C03647=1205.474,-109.246,-38.036,179.217,5.484,149.197
C03648=1205.479,-109.496,-38.027,179.214,5.484,149.197
C03649=1205.485,-109.746,-38.017,179.213,5.484,149.198
C03650=1205.489,-109.996,-38.007,179.210,5.483,149.198
C03651=1205.495,-110.246,-37.997,179.208,5.484,149.199
C03652=1205.501,-110.495,-37.987,179.205,5.483,149.200
C03653=1205.506,-110.745,-37.978,179.203,5.483,149.200
C03654=1205.512,-110.995,-37.968,179.201,5.483,149.201
C03655=1205.516,-111.244,-37.959,179.199,5.483,149.202
C03656=1205.522,-111.495,-37.949,179.196,5.482,149.202
C03657=1205.527,-111.744,-37.939,179.194,5.483,149.203
C03658=1205.532,-111.994,-37.929,179.192,5.482,149.204
C03659=1205.537,-112.244,-37.920,179.190,5.482,149.204
C03660=1205.543,-112.493,-37.910,179.187,5.482,149.205
C03661=1205.549,-112.743,-37.900,179.185,5.482,149.206
C03662=1205.553,-112.993,-37.890,179.183,5.483,149.206
C03663=1205.559,-113.243,-37.880,179.181,5.482,149.207
C03664=1205.564,-113.493,-37.871,179.179,5.482,149.208
C03665=1205.569,-113.742,-37.861,179.176,5.482,149.208
C03666=1205.575,-113.992,-37.852,179.175,5.482,149.209
C03667=1205.580,-114.242,-37.842,179.172,5.482,149.209
C03668=1205.585,-114.491,-37.833,179.170,5.482,149.210
C03669=1205.590,-114.742,-37.822,179.168,5.481,149.211
C03670=1205.596,-114.992,-37.813,179.166,5.482,149.211
C03671=1205.601,-115.241,-37.803,179.163,5.481,149.212
C03672=1205.606,-115.490,-37.794,179.161,5.482,149.213
C03673=1205.611,-115.740,-37.785,179.159,5.481,149.213
C03674=1205.617,-115.990,-37.775,179.157,5.481,149.214
C03675=1205.622,-116.240,-37.766,179.154,5.481,149.215
C03676=1205.628,-116.489,-37.755,179.152,5.481,149.215
C03677=1205.633,-116.739,-37.747,179.150,5.480,149.216
C03678=1205.639,-116.989,-37.737,179.148,5.481,149.217
C03679=1205.643,-117.239,-37.727,179.145,5.480,149.217
C03680=1205.649,-117.489,-37.718,179.143,5.480,149.218
C03681=1205.654,-117.738,-37.708,179.141,5.480,149.219
C03682=1205.659,-117.988,-37.699,179.139,5.480,149.219
C03683=1205.664,-118.238,-37.689,179.136,5.480,149.220
C03684=1205.670,-118.488,-37.680,179.134,5.480,149.220
C03685=1205.675,-118.737,-37.670,179.132,5.479,149.221
C03686=1205.680,-118.987,-37.661,179.130,5.480,149.222
C03687=1205.685,-119.237,-37.652,179.128,5.480,149.222
C03688=1205.691,-119.486,-37.642,179.126,5.479,149.223
C03689=1205.696,-119.736,-37.633,179.124,5.480,149.224
C03690=1205.702,-119.986,-37.623,179.121,5.479,149.224
C03691=1205.706,-120.236,-37.613,179.119,5.479,149.225
C03692=1205.712,-120.486,-37.604,179.117,5.479,149.226
C03693=1205.717,-120.736,-37.594,179.115,5.479,149.226
C03694=1205.722,-120.986,-37.585,179.112,5.478,149.227
C03695=1205.727,-121.235,-37.576,179.110,5.479,149.227
C03696=1205.733,-121.485,-37.566,179.108,5.478,149.228
C03697=1205.738,-121.735,-37.557,179.106,5.478,149.229
C03698=1205.743,-121.984,-37.548,179.103,5.478,149.229
C03699=1205.749,-122.234,-37.538,179.101,5.478,149.230
C03700=1205.754,-122.484,-37.529,179.099,5.478,149.231
C03701=1205.759,-122.733,-37.520,179.097,5.478,149.231
C03702=1205.765,-122.984,-37.510,179.095,5.478,149.232
C03703=1205.770,-123.233,-37.501,179.093,5.478,149.232
C03704=1205.775,-123.483,-37.492,179.091,5.478,149.233
C03705=1205.781,-123.733,-37.482,179.088,5.478,149.234
C03706=1205.786,-123.983,-37.473,179.086,5.478,149.234
C03707=1205.791,-124.232,-37.464,179.084,5.477,149.235
C03708=1205.797,-124.482,-37.454,179.082,5.478,149.236
C03709=1205.802,-124.732,-37.445,179.079,5.477,149.236
C03710=1205.807,-124.982,-37.436,179.077,5.477,149.237
C03711=1205.812,-125.231,-37.427,179.075,5.477,149.238
C03712=1205.818,-125.481,-37.417,179.073,5.477,149.238
C03713=1205.823,-125.731,-37.408,179.070,5.476,149.239
C03714=1205.828,-125.981,-37.400,179.068,5.477,149.240
C03715=1205.834,-126.230,-37.389,179.067,5.477,149.240
C03716=1205.839,-126.480,-37.380,179.064,5.476,149.241
C03717=1205.844,-126.730,-37.372,179.062,5.476,149.241
C03718=1205.423,-126.740,-37.410,179.058,5.480,149.243
C03719=1205.417,-126.491,-37.418,179.060,5.480,149.243
C03720=1205.413,-126.241,-37.428,179.063,5.480,149.242
C03721=1205.407,-125.991,-37.437,179.064,5.480,149.242
C03722=1205.402,-125.741,-37.446,179.066,5.480,149.241
C03723=1205.396,-125.491,-37.455,179.069,5.480,149.240
C03724=1205.391,-125.242,-37.465,179.071,5.480,149.240
C03725=1205.386,-124.992,-37.474,179.073,5.480,149.239
C03726=1205.380,-124.742,-37.483,179.075,5.480,149.238
C03727=1205.375,-124.492,-37.492,179.078,5.481,149.238
C03728=1205.370,-124.243,-37.502,179.080,5.480,149.237
C03729=1205.364,-123.993,-37.511,179.082,5.481,149.236
C03730=1205.359,-123.743,-37.520,179.084,5.481,149.236
C03731=1205.354,-123.494,-37.530,179.087,5.481,149.235
C03732=1205.349,-123.244,-37.539,179.088,5.481,149.235
C03733=1205.343,-122.994,-37.548,179.091,5.482,149.234
C03734=1205.338,-122.744,-37.557,179.093,5.481,149.233
C03735=1205.333,-122.495,-37.567,179.095,5.481,149.233
C03736=1205.327,-122.245,-37.576,179.097,5.482,149.232
C03737=1205.322,-121.995,-37.585,179.099,5.481,149.231
C03738=1205.317,-121.746,-37.595,179.102,5.482,149.231
C03739=1205.312,-121.495,-37.604,179.104,5.482,149.230
C03740=1205.307,-121.246,-37.614,179.106,5.482,149.229
C03741=1205.301,-120.996,-37.623,179.108,5.482,149.229
C03742=1205.296,-120.746,-37.632,179.111,5.482,149.228
C03743=1205.291,-120.497,-37.642,179.112,5.482,149.228
C03744=1205.285,-120.247,-37.651,179.115,5.483,149.227
C03745=1205.280,-119.997,-37.660,179.117,5.482,149.226
C03746=1205.275,-119.748,-37.670,179.119,5.483,149.226
C03747=1205.269,-119.498,-37.679,179.121,5.483,149.225
C03748=1205.264,-119.248,-37.689,179.124,5.483,149.224
C03749=1205.258,-118.998,-37.699,179.126,5.483,149.224
C03750=1205.253,-118.748,-37.707,179.128,5.483,149.223
C03751=1205.249,-118.498,-37.717,179.130,5.483,149.222
C03752=1205.243,-118.248,-37.727,179.132,5.483,149.222
C03753=1205.238,-117.999,-37.736,179.135,5.483,149.221
C03754=1205.232,-117.749,-37.746,179.137,5.483,149.220
C03755=1205.227,-117.500,-37.756,179.139,5.483,149.220
C03756=1205.222,-117.250,-37.765,179.141,5.484,149.219
C03757=1205.216,-117.000,-37.775,179.144,5.484,149.218
C03758=1205.211,-116.750,-37.784,179.146,5.484,149.218
C03759=1205.205,-116.500,-37.793,179.148,5.484,149.217
C03760=1205.200,-116.251,-37.803,179.150,5.484,149.217
C03761=1205.195,-116.001,-37.812,179.153,5.484,149.216
C03762=1205.190,-115.751,-37.822,179.154,5.484,149.215
C03763=1205.185,-115.501,-37.831,179.157,5.485,149.215
C03764=1205.180,-115.251,-37.841,179.159,5.484,149.214
C03765=1205.174,-115.002,-37.850,179.161,5.485,149.213
C03766=1205.169,-114.752,-37.860,179.163,5.485,149.213
C03767=1205.164,-114.503,-37.870,179.166,5.485,149.212
C03768=1205.158,-114.253,-37.880,179.168,5.485,149.212
C03769=1205.153,-114.003,-37.889,179.170,5.486,149.211
C03770=1205.148,-113.753,-37.899,179.172,5.485,149.210
C03771=1205.143,-113.503,-37.909,179.175,5.486,149.209
C03772=1205.137,-113.253,-37.918,179.177,5.486,149.209
C03773=1205.132,-113.004,-37.928,179.179,5.486,149.208
C03774=1205.126,-112.754,-37.937,179.181,5.486,149.207
C03775=1205.121,-112.505,-37.947,179.184,5.486,149.207
C03776=1205.116,-112.255,-37.957,179.186,5.486,149.206
C03777=1205.111,-112.004,-37.966,179.188,5.486,149.206
C03778=1205.106,-111.755,-37.976,179.190,5.486,149.205
C03779=1205.100,-111.505,-37.986,179.193,5.487,149.204
C03780=1205.095,-111.255,-37.996,179.195,5.486,149.204
C03781=1205.089,-111.006,-38.006,179.197,5.486,149.203
C03782=1205.084,-110.756,-38.015,179.199,5.487,149.202
C03783=1205.079,-110.506,-38.025,179.201,5.486,149.202
C03784=1205.074,-110.257,-38.035,179.204,5.487,149.201
C03785=1205.068,-110.006,-38.044,179.205,5.487,149.201
C03786=1205.064,-109.757,-38.054,179.208,5.487,149.200
C03787=1205.058,-109.508,-38.064,179.210,5.487,149.199
C03788=1205.052,-109.258,-38.074,179.212,5.488,149.199
C03789=1205.048,-109.008,-38.084,179.214,5.487,149.198
C03790=1205.042,-108.758,-38.094,179.217,5.488,149.197
C03791=1205.037,-108.508,-38.103,179.219,5.487,149.196
C03792=1205.031,-108.259,-38.113,179.221,5.488,149.196
C03793=1205.026,-108.009,-38.123,179.223,5.488,149.195
C03794=1205.021,-107.759,-38.132,179.226,5.488,149.195
C03795=1205.016,-107.509,-38.143,179.228,5.488,149.194
C03796=1205.011,-107.260,-38.152,179.230,5.488,149.193
C03797=1205.005,-107.010,-38.162,179.233,5.488,149.193
C03798=1205.000,-106.759,-38.172,179.235,5.488,149.192
C03799=1204.995,-106.510,-38.182,179.237,5.488,149.191
C03800=1204.989,-106.261,-38.192,179.239,5.489,149.191
C03801=1204.984,-106.010,-38.202,179.242,5.489,149.190
C03802=1204.979,-105.760,-38.212,179.244,5.489,149.190
C03803=1204.974,-105.511,-38.222,179.246,5.489,149.189
C03804=1204.968,-105.261,-38.232,179.249,5.489,149.188
C03805=1204.963,-105.012,-38.242,179.251,5.489,149.187
C03806=1204.957,-104.762,-38.251,179.253,5.490,149.187
C03807=1204.953,-104.512,-38.261,179.255,5.489,149.186
C03808=1204.947,-104.263,-38.271,179.258,5.490,149.185
C03809=1204.942,-104.013,-38.282,179.260,5.489,149.185
C03810=1204.937,-103.763,-38.292,179.262,5.490,149.184
C03811=1204.932,-103.513,-38.301,179.264,5.490,149.184
C03812=1204.926,-103.263,-38.311,179.267,5.490,149.183
C03813=1204.920,-103.014,-38.321,179.269,5.490,149.182
C03814=1204.916,-102.764,-38.331,179.271,5.491,149.182
C03815=1204.911,-102.514,-38.342,179.273,5.490,149.181
C03816=1204.905,-102.265,-38.352,179.276,5.491,149.180
C03817=1204.901,-102.015,-38.362,179.278,5.491,149.180
C03818=1204.895,-101.765,-38.371,179.280,5.491,149.179
C03819=1204.889,-101.493,-38.383,179.283,5.491,149.178
C03820=1204.883,-101.222,-38.393,179.285,5.491,149.178
C03821=1204.878,-100.951,-38.404,179.287,5.492,149.177
C03822=1204.872,-100.680,-38.416,179.290,5.492,149.176
C03823=1204.867,-100.430,-38.426,179.292,5.492,149.175
C03824=1204.861,-100.180,-38.435,179.295,5.492,149.175
C03825=1204.856,-99.930,-38.446,179.296,5.492,149.174
C03826=1204.851,-99.680,-38.456,179.299,5.492,149.174
C03827=1204.846,-99.431,-38.465,179.301,5.492,149.173
C03828=1204.841,-99.181,-38.476,179.304,5.492,149.172
C03829=1204.835,-98.931,-38.486,179.305,5.492,149.172
C03830=1204.830,-98.682,-38.496,179.308,5.493,149.171
C03831=1204.825,-98.432,-38.507,179.310,5.492,149.170
C03832=1204.820,-98.182,-38.517,179.313,5.493,149.170
C03833=1204.814,-97.933,-38.527,179.314,5.493,149.169
C03834=1204.809,-97.683,-38.537,179.317,5.493,149.168
C03835=1204.804,-97.433,-38.548,179.319,5.493,149.168
C03836=1204.798,-97.183,-38.558,179.322,5.493,149.167
C03837=1204.794,-96.934,-38.568,179.324,5.493,149.166
C03838=1204.788,-96.684,-38.578,179.326,5.494,149.166
C03839=1204.783,-96.434,-38.588,179.328,5.493,149.165
C03840=1204.778,-96.184,-38.599,179.331,5.494,149.164
C03841=1204.772,-95.935,-38.609,179.333,5.494,149.164
C03842=1204.766,-95.685,-38.619,179.335,5.494,149.163
C03843=1204.761,-95.435,-38.630,179.338,5.495,149.162
C03844=1204.756,-95.186,-38.639,179.340,5.494,149.162
C03845=1204.751,-94.935,-38.650,179.342,5.495,149.161
C03846=1204.746,-94.686,-38.660,179.344,5.495,149.160
C03847=1204.740,-94.436,-38.670,179.347,5.495,149.160
C03848=1204.735,-94.186,-38.681,179.349,5.495,149.159
C03849=1204.730,-93.937,-38.691,179.351,5.496,149.159
C03850=1204.725,-93.687,-38.702,179.353,5.495,149.158
C03851=1204.720,-93.438,-38.712,179.356,5.496,149.157
C03852=1204.715,-93.188,-38.722,179.358,5.495,149.156
C03853=1204.710,-92.938,-38.733,179.360,5.496,149.156
C03854=1204.704,-92.688,-38.743,179.362,5.496,149.155
C03855=1204.699,-92.438,-38.754,179.365,5.496,149.155
C03856=1204.693,-92.189,-38.764,179.367,5.496,149.154
C03857=1204.688,-91.939,-38.774,179.370,5.496,149.153
C03858=1204.683,-91.689,-38.785,179.372,5.497,149.153
C03859=1204.677,-91.440,-38.796,179.374,5.496,149.152
C03860=1204.672,-91.190,-38.806,179.377,5.497,149.151
C03861=1204.667,-90.940,-38.816,179.379,5.497,149.150
C03862=1204.662,-90.690,-38.827,179.381,5.497,149.150
C03863=1204.656,-90.440,-38.837,179.383,5.497,149.149
C03864=1204.651,-90.191,-38.847,179.386,5.497,149.149
C03865=1204.647,-89.941,-38.858,179.388,5.497,149.148
C03866=1204.641,-89.692,-38.868,179.390,5.498,149.147
C03867=1204.636,-89.442,-38.879,179.392,5.497,149.147
C03868=1204.631,-89.192,-38.889,179.395,5.498,149.146
C03869=1204.626,-88.942,-38.900,179.397,5.497,149.145
C03870=1204.620,-88.693,-38.910,179.400,5.498,149.145
C03871=1204.615,-88.443,-38.921,179.402,5.499,149.144
C03872=1204.610,-88.193,-38.931,179.404,5.498,149.143
C03873=1204.605,-87.943,-38.942,179.406,5.499,149.143
C03874=1204.599,-87.694,-38.953,179.409,5.498,149.142
C03875=1204.594,-87.444,-38.963,179.411,5.499,149.141
C03876=1204.589,-87.194,-38.974,179.413,5.499,149.141
C03877=1204.584,-86.945,-38.985,179.416,5.499,149.140
C03878=1204.578,-86.695,-38.995,179.418,5.499,149.139
C03879=1204.573,-86.445,-39.006,179.420,5.499,149.139
C03880=1204.568,-86.195,-39.016,179.422,5.499,149.138
C03881=1204.563,-85.946,-39.027,179.425,5.500,149.137
C03882=1204.558,-85.696,-39.037,179.427,5.500,149.137
C03883=1204.553,-85.446,-39.048,179.429,5.500,149.136
C03884=1204.547,-85.197,-39.059,179.432,5.500,149.135
C03885=1204.542,-84.947,-39.069,179.434,5.500,149.135
C03886=1204.536,-84.697,-39.080,179.436,5.501,149.134
C03887=1204.531,-84.447,-39.092,179.438,5.500,149.133
C03888=1204.526,-84.198,-39.102,179.441,5.501,149.133
C03889=1204.521,-83.947,-39.112,179.443,5.500,149.132
C03890=1204.515,-83.698,-39.123,179.445,5.501,149.131
C03891=1204.510,-83.448,-39.134,179.448,5.502,149.131
C03892=1204.505,-83.199,-39.144,179.450,5.501,149.130
C03893=1204.500,-82.949,-39.155,179.453,5.502,149.129
C03894=1204.494,-82.699,-39.166,179.454,5.502,149.129
C03895=1204.490,-82.450,-39.177,179.457,5.502,149.128
C03896=1204.484,-82.200,-39.187,179.459,5.502,149.127
C03897=1204.479,-81.950,-39.198,179.462,5.502,149.127
C03898=1204.474,-81.700,-39.209,179.464,5.503,149.126
C03899=1204.468,-81.451,-39.220,179.466,5.503,149.126
C03900=1204.463,-81.201,-39.231,179.469,5.503,149.125
C03901=1204.458,-80.951,-39.241,179.471,5.503,149.124
C03902=1204.453,-80.702,-39.252,179.473,5.503,149.123
C03903=1204.448,-80.452,-39.263,179.476,5.503,149.123
C03904=1204.443,-80.203,-39.274,179.478,5.504,149.122
C03905=1204.437,-79.952,-39.285,179.480,5.503,149.122
C03906=1204.432,-79.703,-39.295,179.482,5.504,149.121
C03907=1204.427,-79.453,-39.307,179.485,5.504,149.120
C03908=1204.421,-79.203,-39.317,179.487,5.504,149.119
C03909=1204.417,-78.954,-39.328,179.489,5.504,149.119
C03910=1204.412,-78.703,-39.339,179.491,5.504,149.118
C03911=1204.406,-78.454,-39.350,179.494,5.504,149.118
C03912=1204.401,-78.204,-39.361,179.496,5.504,149.117
C03913=1204.395,-77.955,-39.372,179.499,5.505,149.116
C03914=1204.390,-77.705,-39.382,179.501,5.505,149.116
C03915=1204.386,-77.455,-39.394,179.503,5.505,149.115
C03916=1204.380,-77.206,-39.405,179.506,5.505,149.114
C03917=1204.375,-76.956,-39.416,179.508,5.505,149.113
C03918=1204.369,-76.707,-39.427,179.511,5.506,149.113
C03919=1204.364,-76.457,-39.437,179.513,5.506,149.112
C03920=1204.359,-76.207,-39.449,179.515,5.506,149.112
C03921=1204.353,-75.957,-39.459,179.518,5.506,149.111
C03922=1204.349,-75.707,-39.471,179.520,5.506,149.110
C03923=1204.343,-75.436,-39.483,179.522,5.506,149.109
C03924=1204.337,-75.166,-39.495,179.525,5.507,149.109
C03925=1204.332,-74.896,-39.506,179.527,5.507,149.108
C03926=1204.326,-74.625,-39.518,179.530,5.507,149.107
C03927=1204.321,-74.375,-39.529,179.532,5.507,149.107
C03928=1204.315,-74.125,-39.541,179.534,5.507,149.106
C03929=1204.310,-73.876,-39.552,179.537,5.507,149.105
C03930=1204.305,-73.626,-39.562,179.539,5.507,149.105
C03931=1204.300,-73.376,-39.573,179.541,5.508,149.104
C03932=1204.294,-73.127,-39.585,179.544,5.508,149.103
C03933=1204.289,-72.877,-39.596,179.546,5.508,149.103
C03934=1204.284,-72.627,-39.607,179.549,5.508,149.102
C03935=1204.278,-72.378,-39.618,179.550,5.508,149.101
C03936=1204.273,-72.128,-39.629,179.553,5.509,149.101
C03937=1204.269,-71.878,-39.640,179.556,5.509,149.100
C03938=1204.263,-71.629,-39.652,179.558,5.509,149.099
C03939=1204.258,-71.379,-39.662,179.561,5.509,149.099
C03940=1204.253,-71.129,-39.674,179.563,5.509,149.098
C03941=1204.248,-70.879,-39.686,179.565,5.510,149.097
C03942=1204.242,-70.630,-39.696,179.567,5.510,149.097
C03943=1204.237,-70.380,-39.707,179.570,5.510,149.096
C03944=1204.232,-70.130,-39.719,179.572,5.510,149.095
C03945=1204.227,-69.881,-39.730,179.574,5.510,149.095
C03946=1204.222,-69.631,-39.741,179.577,5.510,149.094
C03947=1204.216,-69.381,-39.752,179.579,5.511,149.093
C03948=1204.211,-69.131,-39.764,179.581,5.511,149.093
C03949=1204.205,-68.882,-39.775,179.584,5.511,149.092
C03950=1204.201,-68.632,-39.786,179.586,5.511,149.091
C03951=1204.196,-68.382,-39.797,179.589,5.511,149.091
C03952=1204.190,-68.133,-39.808,179.591,5.512,149.090
C03953=1204.185,-67.883,-39.820,179.593,5.512,149.089
C03954=1204.180,-67.633,-39.832,179.596,5.512,149.089
C03955=1204.175,-67.384,-39.843,179.598,5.512,149.088
C03956=1204.169,-67.134,-39.853,179.600,5.512,149.087
C03957=1204.164,-66.884,-39.865,179.603,5.513,149.087
C03958=1204.159,-66.635,-39.876,179.605,5.513,149.086
C03959=1204.154,-66.385,-39.888,179.607,5.513,149.085
C03960=1204.149,-66.135,-39.900,179.609,5.513,149.085
C03961=1204.143,-65.886,-39.911,179.612,5.513,149.084
C03962=1204.138,-65.636,-39.922,179.615,5.514,149.083
C03963=1204.133,-65.386,-39.933,179.617,5.513,149.083
C03964=1204.128,-65.136,-39.945,179.619,5.514,149.082
C03965=1204.123,-64.887,-39.956,179.621,5.514,149.081
C03966=1204.117,-64.637,-39.968,179.624,5.514,149.081
C03967=1204.113,-64.387,-39.979,179.626,5.515,149.080
C03968=1204.107,-64.138,-39.991,179.628,5.514,149.079
C03969=1204.102,-63.888,-40.002,179.631,5.515,149.079
C03970=1204.096,-63.639,-40.014,179.633,5.516,149.078
C03971=1204.092,-63.389,-40.025,179.635,5.515,149.077
C03972=1204.086,-63.139,-40.037,179.638,5.516,149.077
C03973=1204.082,-62.889,-40.048,179.640,5.515,149.076
C03974=1204.076,-62.640,-40.060,179.643,5.516,149.075
C03975=1204.071,-62.391,-40.071,179.646,5.516,149.075
C03976=1204.065,-62.141,-40.083,179.647,5.516,149.074
C03977=1204.061,-61.891,-40.094,179.650,5.517,149.073
C03978=1204.055,-61.640,-40.105,179.652,5.517,149.073
C03979=1204.050,-61.391,-40.116,179.655,5.517,149.072
C03980=1204.045,-61.141,-40.128,179.657,5.517,149.071
C03981=1204.040,-60.892,-40.139,179.659,5.517,149.071
C03982=1204.034,-60.643,-40.152,179.661,5.518,149.070
C03983=1204.030,-60.393,-40.163,179.664,5.518,149.069
C03984=1204.024,-60.143,-40.175,179.666,5.518,149.069
C03985=1204.019,-59.893,-40.187,179.669,5.518,149.068
C03986=1204.014,-59.644,-40.198,179.672,5.519,149.067
C03987=1204.009,-59.394,-40.210,179.674,5.518,149.067
C03988=1204.003,-59.145,-40.221,179.676,5.519,149.066
C03989=1203.998,-58.895,-40.233,179.678,5.519,149.065
C03990=1203.993,-58.645,-40.244,179.681,5.519,149.065
C03991=1203.988,-58.395,-40.256,179.683,5.520,149.064
C03992=1203.982,-58.145,-40.268,179.685,5.519,149.063
C03993=1203.978,-57.896,-40.279,179.688,5.520,149.063
C03994=1203.972,-57.646,-40.291,179.691,5.520,149.062
C03995=1203.968,-57.396,-40.302,179.692,5.520,149.061
C03996=1203.962,-57.146,-40.314,179.695,5.521,149.061
C03997=1203.957,-56.898,-40.327,179.698,5.521,149.060
C03998=1203.952,-56.648,-40.338,179.700,5.521,149.059
C03999=1203.946,-56.398,-40.350,179.702,5.521,149.059
C04000=1203.942,-56.148,-40.361,179.704,5.521,149.058
C04001=1203.936,-55.898,-40.373,179.707,5.522,149.057
C04002=1203.931,-55.648,-40.385,179.709,5.522,149.057
C04003=1203.926,-55.399,-40.396,179.711,5.522,149.056
C04004=1203.921,-55.150,-40.409,179.714,5.522,149.055
C04005=1203.916,-54.900,-40.421,179.717,5.523,149.055
C04006=1203.911,-54.650,-40.432,179.719,5.522,149.054
C04007=1203.905,-54.400,-40.444,179.721,5.523,149.053
C04008=1203.900,-54.150,-40.456,179.724,5.524,149.053
C04009=1203.896,-53.901,-40.468,179.726,5.523,149.052
C04010=1203.890,-53.651,-40.480,179.728,5.524,149.051
C04011=1203.884,-53.402,-40.491,179.731,5.524,149.051
C04012=1203.880,-53.152,-40.502,179.733,5.524,149.050
C04013=1203.874,-52.903,-40.515,179.736,5.524,149.049
C04014=1203.869,-52.653,-40.527,179.738,5.525,149.049
C04015=1203.864,-52.403,-40.539,179.740,5.525,149.048
C04016=1203.859,-52.153,-40.550,179.743,5.525,149.047
C04017=1203.854,-51.904,-40.563,179.745,5.526,149.047
C04018=1203.848,-51.654,-40.574,179.747,5.525,149.046
C04019=1203.844,-51.405,-40.586,179.750,5.526,149.045
C04020=1203.838,-51.155,-40.598,179.753,5.526,149.044
C04021=1203.833,-50.905,-40.610,179.754,5.526,149.044
C04022=1203.828,-50.655,-40.622,179.757,5.527,149.043
C04023=1203.822,-50.405,-40.634,179.759,5.526,149.043
C04024=1203.818,-50.156,-40.646,179.762,5.527,149.042
C04025=1203.812,-49.907,-40.658,179.764,5.527,149.041
C04026=1203.807,-49.657,-40.670,179.767,5.527,149.040
C04027=1203.802,-49.386,-40.683,179.769,5.527,149.040
C04028=1203.796,-49.117,-40.696,179.772,5.528,149.039
C04029=1203.791,-48.847,-40.709,179.775,5.528,149.038
C04030=1203.785,-48.576,-40.722,179.777,5.529,149.038
C04031=1203.780,-48.327,-40.734,179.779,5.528,149.037
C04032=1203.775,-48.077,-40.747,179.782,5.529,149.036
C04033=1203.769,-47.827,-40.758,179.785,5.529,149.036
C04034=1203.764,-47.577,-40.770,179.786,5.529,149.035
C04035=1203.760,-47.328,-40.782,179.789,5.530,149.034
C04036=1203.754,-47.078,-40.794,179.792,5.530,149.034
C04037=1203.749,-46.829,-40.807,179.794,5.530,149.033
C04038=1203.744,-46.579,-40.819,179.796,5.530,149.032
C04039=1203.738,-46.329,-40.831,179.799,5.531,149.032
C04040=1203.733,-46.080,-40.843,179.801,5.531,149.031
C04041=1203.728,-45.830,-40.854,179.803,5.531,149.030
C04042=1203.723,-45.581,-40.867,179.806,5.532,149.030
C04043=1203.718,-45.331,-40.879,179.808,5.531,149.029
C04044=1203.713,-45.082,-40.892,179.811,5.532,149.028
C04045=1203.707,-44.832,-40.903,179.813,5.532,149.028
C04046=1203.702,-44.582,-40.916,179.816,5.533,149.027
C04047=1203.697,-44.333,-40.928,179.818,5.533,149.026
C04048=1203.692,-44.083,-40.940,179.820,5.533,149.026
C04049=1203.686,-43.833,-40.952,179.823,5.534,149.025
C04050=1203.682,-43.584,-40.965,179.825,5.533,149.024
C04051=1203.677,-43.334,-40.977,179.828,5.534,149.024
C04052=1203.672,-43.084,-40.989,179.830,5.534,149.023
C04053=1203.666,-42.834,-41.001,179.832,5.534,149.022
C04054=1203.661,-42.585,-41.014,179.835,5.534,149.021
C04055=1203.656,-42.335,-41.026,179.837,5.535,149.021
C04056=1203.651,-42.086,-41.038,179.839,5.535,149.020
C04057=1203.645,-41.836,-41.050,179.842,5.535,149.020
C04058=1203.640,-41.587,-41.063,179.845,5.536,149.019
C04059=1203.635,-41.337,-41.075,179.847,5.536,149.018
C04060=1203.630,-41.087,-41.088,179.849,5.536,149.017
C04061=1203.625,-40.837,-41.100,179.852,5.536,149.017
C04062=1203.620,-40.587,-41.112,179.854,5.537,149.016
C04063=1203.615,-40.338,-41.125,179.856,5.537,149.016
C04064=1203.609,-40.089,-41.137,179.859,5.537,149.015
C04065=1203.604,-39.839,-41.149,179.862,5.538,149.014
C04066=1203.599,-39.589,-41.162,179.864,5.538,149.014
C04067=1203.593,-39.340,-41.174,179.866,5.538,149.013
C04068=1203.589,-39.089,-41.187,179.869,5.538,149.012
C04069=1203.584,-38.840,-41.199,179.871,5.539,149.012
C04070=1203.578,-38.590,-41.211,179.873,5.539,149.011
C04071=1203.573,-38.341,-41.224,179.876,5.539,149.010
C04072=1203.568,-38.092,-41.236,179.879,5.540,149.010
C04073=1203.563,-37.842,-41.248,179.881,5.540,149.009
C04074=1203.558,-37.592,-41.261,179.883,5.540,149.008
C04075=1203.553,-37.342,-41.274,179.886,5.541,149.007
C04076=1203.548,-37.092,-41.286,179.888,5.541,149.007
C04077=1203.542,-36.843,-41.298,179.890,5.541,149.006
C04078=1203.537,-36.594,-41.311,179.893,5.541,149.006
C04079=1203.532,-36.344,-41.323,179.896,5.542,149.005
C04080=1203.527,-36.094,-41.336,179.898,5.542,149.004
C04081=1203.522,-35.844,-41.348,179.900,5.542,149.003
C04082=1203.517,-35.595,-41.361,179.903,5.543,149.003
C04083=1203.512,-35.346,-41.373,179.905,5.543,149.002
C04084=1203.507,-35.096,-41.385,179.907,5.543,149.002
C04085=1203.502,-34.846,-41.398,179.910,5.544,149.001
C04086=1203.496,-34.596,-41.412,179.913,5.544,149.000
C04087=1203.491,-34.347,-41.424,179.915,5.544,149.000
C04088=1203.486,-34.097,-41.436,179.917,5.544,148.999
C04089=1203.481,-33.848,-41.449,179.920,5.545,148.998
C04090=1203.476,-33.598,-41.462,179.922,5.545,148.998
C04091=1203.471,-33.348,-41.474,179.924,5.545,148.997
C04092=1203.466,-33.099,-41.487,179.927,5.546,148.996
C04093=1203.461,-32.850,-41.499,179.930,5.546,148.996
C04094=1203.455,-32.599,-41.512,179.932,5.546,148.995
C04095=1203.450,-32.349,-41.525,179.934,5.546,148.994
C04096=1203.445,-32.100,-41.537,179.937,5.547,148.993
C04097=1203.440,-31.851,-41.550,179.939,5.547,148.993
C04098=1203.435,-31.601,-41.563,179.941,5.547,148.992
C04099=1203.430,-31.351,-41.576,179.944,5.548,148.992
C04100=1203.425,-31.102,-41.588,179.947,5.548,148.991
C04101=1203.419,-30.852,-41.601,179.949,5.548,148.990
C04102=1203.414,-30.602,-41.614,179.951,5.548,148.989
C04103=1203.409,-30.353,-41.626,179.954,5.549,148.989
C04104=1203.404,-30.103,-41.639,179.957,5.549,148.988
C04105=1203.399,-29.854,-41.651,179.958,5.549,148.988
C04106=1203.394,-29.604,-41.665,179.961,5.550,148.987
C04107=1203.388,-29.354,-41.678,179.963,5.550,148.986
C04108=1203.383,-29.105,-41.690,179.966,5.551,148.986
C04109=1203.379,-28.855,-41.703,179.968,5.550,148.985
C04110=1203.374,-28.606,-41.716,179.971,5.551,148.984
C04111=1203.368,-28.356,-41.729,179.974,5.551,148.983
C04112=1203.363,-28.107,-41.742,179.976,5.552,148.983
C04113=1203.358,-27.857,-41.755,179.978,5.552,148.982
C04114=1203.353,-27.607,-41.767,179.980,5.552,148.982
C04115=1203.347,-27.358,-41.780,179.983,5.553,148.981
C04116=1203.343,-27.108,-41.793,179.986,5.553,148.980
C04117=1203.338,-26.858,-41.806,179.988,5.553,148.979
C04118=1203.332,-26.609,-41.818,179.991,5.553,148.979
C04119=1203.327,-26.359,-41.832,179.993,5.554,148.978
C04120=1203.322,-26.109,-41.845,179.995,5.555,148.978
C04121=1203.317,-25.860,-41.857,179.997,5.554,148.977
C04122=1203.312,-25.610,-41.871,-180.000,5.555,148.976
C04123=1203.307,-25.360,-41.883,-179.997,5.555,148.976
C04124=1203.301,-25.111,-41.896,-179.995,5.556,148.975
C04125=1203.297,-24.861,-41.909,-179.993,5.555,148.974
C04126=1203.291,-24.612,-41.922,-179.990,5.556,148.974
C04127=1203.286,-24.362,-41.935,-179.988,5.557,148.973
C04128=1203.281,-24.112,-41.948,-179.985,5.557,148.972
C04129=1203.276,-23.863,-41.962,-179.983,5.557,148.972
C04130=1203.271,-23.613,-41.975,-179.980,5.557,148.971
C04131=1203.265,-23.344,-41.989,-179.978,5.558,148.970
C04132=1203.260,-23.074,-42.002,-179.975,5.558,148.970
C04133=1203.254,-22.804,-42.016,-179.972,5.559,148.969
C04134=1203.249,-22.536,-42.031,-179.970,5.559,148.968
C04135=1203.244,-22.285,-42.044,-179.967,5.560,148.967
C04136=1203.239,-22.036,-42.057,-179.965,5.559,148.967
C04137=1203.234,-21.786,-42.070,-179.962,5.560,148.966
C04138=1203.228,-21.536,-42.083,-179.960,5.560,148.965
C04139=1203.223,-21.288,-42.096,-179.957,5.561,148.965
C04140=1203.218,-21.037,-42.110,-179.955,5.561,148.964
C04141=1203.213,-20.788,-42.122,-179.953,5.561,148.963
C04142=1203.208,-20.538,-42.135,-179.950,5.562,148.963
C04143=1203.203,-20.288,-42.148,-179.947,5.562,148.962
C04144=1203.198,-20.040,-42.162,-179.945,5.562,148.961
C04145=1203.193,-19.789,-42.175,-179.943,5.562,148.961
C04146=1203.187,-19.540,-42.188,-179.940,5.563,148.960
C04147=1203.183,-19.290,-42.201,-179.938,5.564,148.960
C04148=1203.177,-19.041,-42.215,-179.935,5.564,148.959
C04149=1203.172,-18.792,-42.227,-179.933,5.564,148.958
C04150=1203.167,-18.541,-42.241,-179.930,5.564,148.957
C04151=1203.162,-18.292,-42.254,-179.928,5.565,148.957
C04152=1203.157,-18.042,-42.268,-179.925,5.565,148.956
C04153=1203.152,-17.793,-42.280,-179.923,5.565,148.955
C04154=1203.146,-17.543,-42.294,-179.921,5.566,148.955
C04155=1203.142,-17.294,-42.307,-179.918,5.566,148.954
C04156=1203.136,-17.044,-42.321,-179.916,5.567,148.954
C04157=1203.131,-16.794,-42.334,-179.913,5.567,148.953
C04158=1203.126,-16.545,-42.348,-179.911,5.567,148.952
C04159=1203.121,-16.295,-42.360,-179.908,5.567,148.951
C04160=1203.116,-16.045,-42.374,-179.905,5.568,148.951
C04161=1203.111,-15.796,-42.387,-179.903,5.569,148.950
C04162=1203.105,-15.547,-42.400,-179.901,5.569,148.950
C04163=1203.101,-15.297,-42.413,-179.899,5.569,148.949
C04164=1203.095,-15.048,-42.427,-179.896,5.569,148.948
C04165=1203.091,-14.798,-42.440,-179.893,5.570,148.947
C04166=1203.085,-14.548,-42.454,-179.891,5.570,148.947
C04167=1203.081,-14.299,-42.467,-179.888,5.571,148.946
C04168=1203.075,-14.049,-42.480,-179.886,5.571,148.946
C04169=1203.070,-13.800,-42.494,-179.884,5.571,148.945
C04170=1203.065,-13.550,-42.507,-179.881,5.572,148.944
C04171=1203.060,-13.300,-42.521,-179.878,5.572,148.944
C04172=1203.055,-13.050,-42.535,-179.876,5.573,148.943
C04173=1203.050,-12.801,-42.547,-179.874,5.573,148.942
C04174=1203.045,-12.551,-42.561,-179.871,5.573,148.941
C04175=1203.039,-12.302,-42.575,-179.869,5.574,148.941
C04176=1203.035,-12.052,-42.588,-179.866,5.574,148.940
C04177=1203.029,-11.802,-42.601,-179.863,5.575,148.940
C04178=1203.025,-11.553,-42.615,-179.861,5.575,148.939
C04179=1203.019,-11.303,-42.628,-179.859,5.575,148.938
C04180=1203.014,-11.054,-42.643,-179.856,5.575,148.938
C04181=1203.009,-10.804,-42.655,-179.853,5.576,148.937
C04182=1203.004,-10.555,-42.669,-179.851,5.577,148.936
C04183=1202.999,-10.305,-42.682,-179.849,5.577,148.936
C04184=1202.994,-10.056,-42.696,-179.847,5.577,148.935
C04185=1202.989,-9.805,-42.710,-179.844,5.577,148.934
C04186=1202.984,-9.557,-42.723,-179.841,5.578,148.934
C04187=1202.979,-9.307,-42.738,-179.839,5.578,148.933
C04188=1202.973,-9.057,-42.751,-179.836,5.579,148.932
C04189=1202.969,-8.808,-42.764,-179.834,5.579,148.932
C04190=1202.964,-8.558,-42.778,-179.832,5.579,148.931
C04191=1202.958,-8.309,-42.792,-179.829,5.580,148.930
C04192=1202.953,-8.059,-42.805,-179.826,5.580,148.930
C04193=1202.948,-7.810,-42.819,-179.824,5.581,148.929
C04194=1202.943,-7.560,-42.833,-179.821,5.581,148.928
C04195=1202.938,-7.310,-42.846,-179.819,5.581,148.928
C04196=1202.933,-7.061,-42.860,-179.817,5.582,148.927
C04197=1202.928,-6.811,-42.874,-179.814,5.582,148.926
C04198=1202.923,-6.562,-42.887,-179.812,5.583,148.926
C04199=1202.918,-6.312,-42.901,-179.809,5.583,148.925
C04200=1202.913,-6.062,-42.915,-179.806,5.584,148.924
C04201=1202.907,-5.813,-42.929,-179.804,5.584,148.924
C04202=1202.903,-5.563,-42.942,-179.802,5.584,148.923
C04203=1202.898,-5.314,-42.956,-179.799,5.585,148.923
C04204=1202.892,-5.064,-42.970,-179.797,5.585,148.922
C04205=1202.887,-4.814,-42.984,-179.794,5.586,148.921
C04206=1202.883,-4.565,-42.998,-179.791,5.586,148.921
C04207=1202.877,-4.315,-43.011,-179.789,5.586,148.920
C04208=1202.872,-4.066,-43.025,-179.787,5.587,148.919
C04209=1202.866,-3.817,-43.039,-179.784,5.587,148.919
C04210=1202.862,-3.567,-43.053,-179.782,5.588,148.918
C04211=1202.857,-3.317,-43.066,-179.779,5.588,148.917
C04212=1202.851,-3.068,-43.080,-179.776,5.589,148.917
C04213=1202.846,-2.818,-43.094,-179.774,5.589,148.916
C04214=1202.842,-2.568,-43.109,-179.772,5.589,148.915
C04215=1202.836,-2.319,-43.121,-179.769,5.590,148.915
C04216=1202.831,-2.069,-43.136,-179.767,5.590,148.914
C04217=1202.826,-1.820,-43.150,-179.764,5.591,148.913
C04218=1202.822,-1.570,-43.164,-179.762,5.591,148.913
C04219=1202.816,-1.321,-43.178,-179.759,5.592,148.912
C04220=1202.811,-1.071,-43.191,-179.757,5.592,148.911
C04221=1202.807,-0.821,-43.205,-179.754,5.592,148.911
C04222=1202.801,-0.572,-43.219,-179.752,5.593,148.910
C04223=1202.796,-0.322,-43.234,-179.749,5.594,148.909
C04224=1202.791,-0.073,-43.248,-179.747,5.594,148.909
C04225=1202.785,0.176,-43.262,-179.744,5.595,148.908
C04226=1202.780,0.427,-43.275,-179.741,5.595,148.907
C04227=1202.776,0.676,-43.289,-179.739,5.595,148.907
C04228=1202.771,0.926,-43.303,-179.737,5.596,148.906
C04229=1202.765,1.175,-43.317,-179.735,5.596,148.906
C04230=1202.761,1.424,-43.331,-179.732,5.597,148.905
C04231=1202.756,1.674,-43.346,-179.729,5.597,148.904
C04232=1202.751,1.924,-43.360,-179.727,5.598,148.904
C04233=1202.745,2.173,-43.374,-179.724,5.598,148.903
C04234=1202.740,2.423,-43.388,-179.721,5.599,148.902
C04235=1202.735,2.692,-43.403,-179.719,5.599,148.901
C04236=1202.729,2.961,-43.418,-179.716,5.600,148.901
C04237=1202.724,3.230,-43.434,-179.713,5.600,148.900
C04238=1202.718,3.499,-43.448,-179.711,5.601,148.899
C04239=1202.713,3.749,-43.463,-179.708,5.601,148.899
C04240=1202.708,3.998,-43.477,-179.706,5.601,148.898
C04241=1202.703,4.248,-43.491,-179.704,5.602,148.898
C04242=1202.698,4.498,-43.506,-179.701,5.602,148.897
C04243=1202.693,4.747,-43.520,-179.699,5.603,148.896
C04244=1202.688,4.996,-43.534,-179.696,5.603,148.895
C04245=1202.683,5.246,-43.548,-179.693,5.604,148.895
C04246=1202.678,5.496,-43.562,-179.691,5.604,148.894
C04247=1202.672,5.745,-43.576,-179.688,5.605,148.894
C04248=1202.667,5.995,-43.591,-179.686,5.605,148.893
C04249=1202.662,6.244,-43.605,-179.684,5.605,148.892
C04250=1202.657,6.494,-43.619,-179.681,5.606,148.892
C04251=1202.652,6.744,-43.633,-179.678,5.606,148.891
C04252=1202.648,6.993,-43.648,-179.676,5.607,148.890
C04253=1202.642,7.242,-43.662,-179.674,5.608,148.890
C04254=1202.637,7.492,-43.677,-179.671,5.608,148.889
C04255=1202.632,7.741,-43.691,-179.668,5.609,148.888
C04256=1202.627,7.991,-43.705,-179.666,5.609,148.888
C04257=1202.622,8.241,-43.719,-179.663,5.610,148.887
C04258=1202.618,8.490,-43.734,-179.661,5.610,148.887
C04259=1202.612,8.739,-43.748,-179.659,5.610,148.886
C04260=1202.607,8.989,-43.762,-179.656,5.611,148.885
C04261=1202.602,9.238,-43.777,-179.653,5.611,148.885
C04262=1202.597,9.488,-43.791,-179.651,5.612,148.884
C04263=1202.592,9.738,-43.805,-179.648,5.612,148.883
C04264=1202.587,9.987,-43.820,-179.646,5.613,148.883
C04265=1202.583,10.237,-43.834,-179.643,5.613,148.882
C04266=1202.577,10.486,-43.848,-179.641,5.614,148.881
C04267=1202.572,10.735,-43.863,-179.638,5.614,148.881
C04268=1202.567,10.985,-43.878,-179.635,5.615,148.880
C04269=1202.562,11.235,-43.892,-179.633,5.615,148.879
C04270=1202.557,11.485,-43.906,-179.631,5.616,148.879
C04271=1202.552,11.734,-43.921,-179.628,5.616,148.878
C04272=1202.547,11.983,-43.936,-179.626,5.617,148.877
C04273=1202.542,12.233,-43.950,-179.623,5.617,148.877
C04274=1202.537,12.483,-43.964,-179.621,5.618,148.876
C04275=1202.531,12.732,-43.979,-179.618,5.618,148.876
C04276=1202.526,12.981,-43.994,-179.616,5.619,148.875
C04277=1202.521,13.231,-44.008,-179.613,5.619,148.874
C04278=1202.516,13.481,-44.022,-179.610,5.620,148.874
C04279=1202.512,13.730,-44.037,-179.608,5.620,148.873
C04280=1202.507,13.979,-44.051,-179.605,5.621,148.872
C04281=1202.501,14.229,-44.066,-179.604,5.621,148.872
C04282=1202.496,14.479,-44.081,-179.601,5.622,148.871
C04283=1202.491,14.728,-44.096,-179.598,5.622,148.870
C04284=1202.486,14.978,-44.110,-179.596,5.623,148.870
C04285=1202.482,15.227,-44.125,-179.593,5.623,148.869
C04286=1202.476,15.477,-44.140,-179.590,5.624,148.868
C04287=1202.471,15.727,-44.154,-179.588,5.624,148.868
C04288=1202.467,15.976,-44.169,-179.585,5.625,148.867
C04289=1202.462,16.226,-44.183,-179.583,5.625,148.866
C04290=1202.456,16.475,-44.197,-179.580,5.626,148.866
C04291=1202.451,16.724,-44.213,-179.578,5.626,148.865
C04292=1202.446,16.974,-44.227,-179.575,5.627,148.865
C04293=1202.441,17.223,-44.242,-179.573,5.628,148.864
C04294=1202.436,17.473,-44.256,-179.570,5.628,148.863
C04295=1202.430,17.723,-44.271,-179.567,5.629,148.863
C04296=1202.426,17.972,-44.286,-179.565,5.629,148.862
C04297=1202.421,18.221,-44.300,-179.563,5.629,148.861
C04298=1202.415,18.471,-44.316,-179.561,5.630,148.861
C04299=1202.410,18.720,-44.330,-179.558,5.630,148.860
C04300=1202.406,18.970,-44.345,-179.555,5.631,148.859
C04301=1202.401,19.219,-44.360,-179.553,5.632,148.859
C04302=1202.395,19.469,-44.375,-179.550,5.632,148.858
C04303=1202.391,19.718,-44.389,-179.548,5.633,148.858
C04304=1202.386,19.967,-44.404,-179.545,5.633,148.857
C04305=1202.380,20.217,-44.419,-179.542,5.634,148.856
C04306=1202.376,20.467,-44.434,-179.540,5.634,148.856
C04307=1202.371,20.716,-44.449,-179.537,5.635,148.855
C04308=1202.365,20.966,-44.464,-179.535,5.636,148.854
C04309=1202.361,21.216,-44.479,-179.532,5.636,148.854
C04310=1202.356,21.465,-44.494,-179.530,5.637,148.853
C04311=1202.350,21.715,-44.509,-179.527,5.637,148.852
C04312=1202.346,21.964,-44.524,-179.524,5.638,148.852
C04313=1202.341,22.213,-44.539,-179.522,5.639,148.851
C04314=1202.335,22.463,-44.554,-179.520,5.639,148.851
C04315=1202.331,22.712,-44.569,-179.517,5.640,148.850
C04316=1202.325,22.963,-44.583,-179.514,5.640,148.849
C04317=1202.321,23.212,-44.598,-179.512,5.641,148.849
C04318=1202.316,23.461,-44.613,-179.510,5.642,148.848
C04319=1202.310,23.711,-44.628,-179.507,5.642,148.847
C04320=1202.306,23.960,-44.643,-179.505,5.642,148.847
C04321=1202.300,24.209,-44.659,-179.502,5.642,148.846
C04322=1202.295,24.459,-44.673,-179.500,5.643,148.845
C04323=1202.291,24.708,-44.688,-179.497,5.644,148.845
C04324=1202.286,24.958,-44.704,-179.495,5.644,148.844
C04325=1202.281,25.208,-44.718,-179.492,5.645,148.844
C04326=1202.275,25.457,-44.734,-179.489,5.645,148.843
C04327=1202.271,25.706,-44.749,-179.487,5.646,148.842
C04328=1202.265,25.956,-44.764,-179.485,5.647,148.842
C04329=1202.260,26.205,-44.779,-179.482,5.647,148.841
C04330=1202.255,26.455,-44.794,-179.479,5.648,148.840
C04331=1202.250,26.705,-44.809,-179.477,5.648,148.840
C04332=1202.245,26.954,-44.824,-179.474,5.649,148.839
C04333=1202.241,27.204,-44.840,-179.472,5.650,148.839
C04334=1202.235,27.453,-44.855,-179.469,5.650,148.838
C04335=1202.230,27.703,-44.869,-179.467,5.651,148.837
C04336=1202.225,27.952,-44.885,-179.464,5.651,148.837
C04337=1202.220,28.201,-44.900,-179.461,5.652,148.836
C04338=1202.215,28.451,-44.916,-179.459,5.653,148.835
C04339=1202.210,28.720,-44.931,-179.457,5.653,148.835
C04340=1202.204,28.988,-44.948,-179.453,5.655,148.834
C04341=1202.199,29.257,-44.964,-179.451,5.655,148.833
C04342=1202.193,29.525,-44.981,-179.448,5.656,148.833
C04343=1202.189,29.776,-44.996,-179.445,5.656,148.832
C04344=1202.184,30.025,-45.011,-179.443,5.657,148.831
C04345=1202.178,30.275,-45.027,-179.440,5.657,148.831
C04346=1202.174,30.524,-45.042,-179.438,5.658,148.830
C04347=1202.168,30.773,-45.057,-179.435,5.659,148.830
C04348=1202.164,31.022,-45.072,-179.433,5.659,148.829
C04349=1202.159,31.272,-45.088,-179.430,5.660,148.828
C04350=1202.154,31.522,-45.103,-179.427,5.660,148.828
C04351=1202.149,31.771,-45.118,-179.425,5.661,148.827
C04352=1202.143,32.021,-45.134,-179.423,5.662,148.826
C04353=1202.139,32.270,-45.149,-179.420,5.662,148.826
C04354=1202.134,32.520,-45.165,-179.417,5.663,148.825
C04355=1202.129,32.769,-45.180,-179.415,5.663,148.825
C04356=1202.124,33.018,-45.195,-179.412,5.664,148.824
C04357=1202.118,33.268,-45.211,-179.410,5.664,148.823
C04358=1202.114,33.518,-45.226,-179.407,5.665,148.823
C04359=1202.109,33.767,-45.242,-179.405,5.666,148.822
C04360=1202.103,34.016,-45.258,-179.402,5.666,148.821
C04361=1202.099,34.265,-45.273,-179.400,5.667,148.821
C04362=1202.094,34.516,-45.288,-179.397,5.667,148.820
C04363=1202.089,34.765,-45.304,-179.394,5.668,148.819
C04364=1202.084,35.014,-45.319,-179.392,5.669,148.819
C04365=1202.079,35.263,-45.335,-179.390,5.669,148.818
C04366=1202.074,35.514,-45.351,-179.387,5.670,148.818
C04367=1202.069,35.763,-45.366,-179.384,5.670,148.817
C04368=1202.064,36.012,-45.381,-179.382,5.671,148.816
C04369=1202.058,36.261,-45.397,-179.380,5.672,148.816
C04370=1202.054,36.511,-45.412,-179.377,5.672,148.815
C04371=1202.049,36.761,-45.428,-179.374,5.673,148.814
C04372=1202.044,37.010,-45.443,-179.372,5.673,148.814
C04373=1202.038,37.259,-45.459,-179.370,5.674,148.813
C04374=1202.034,37.509,-45.474,-179.367,5.675,148.813
C04375=1202.029,37.759,-45.490,-179.364,5.676,148.812
C04376=1202.024,38.007,-45.506,-179.361,5.677,148.811
C04377=1202.019,38.258,-45.522,-179.359,5.678,148.811
C04378=1202.014,38.507,-45.537,-179.356,5.678,148.810
C04379=1202.009,38.756,-45.553,-179.354,5.679,148.810
C04380=1202.003,39.005,-45.568,-179.351,5.679,148.809
C04381=1201.999,39.256,-45.584,-179.349,5.680,148.808
C04382=1201.994,39.505,-45.599,-179.346,5.681,148.808
C04383=1201.989,39.753,-45.615,-179.343,5.681,148.807
C04384=1201.984,40.004,-45.631,-179.341,5.682,148.806
C04385=1201.979,40.253,-45.647,-179.339,5.683,148.806
C04386=1201.973,40.502,-45.663,-179.336,5.683,148.805
C04387=1201.969,40.752,-45.678,-179.333,5.684,148.805
C04388=1201.964,41.002,-45.694,-179.331,5.684,148.804
C04389=1201.959,41.250,-45.710,-179.328,5.685,148.803
C04390=1201.954,41.500,-45.726,-179.326,5.686,148.803
C04391=1201.949,41.750,-45.741,-179.323,5.686,148.802
C04392=1201.943,41.999,-45.757,-179.321,5.687,148.801
C04393=1201.940,42.248,-45.773,-179.318,5.687,148.801
C04394=1201.934,42.498,-45.789,-179.315,5.689,148.800
C04395=1201.929,42.748,-45.805,-179.313,5.689,148.800
C04396=1201.924,42.997,-45.820,-179.310,5.690,148.799
C04397=1201.919,43.246,-45.837,-179.307,5.690,148.798
C04398=1201.914,43.496,-45.852,-179.305,5.691,148.798
C04399=1201.909,43.746,-45.868,-179.303,5.692,148.797
C04400=1201.904,43.994,-45.884,-179.300,5.692,148.797
C04401=1201.900,44.244,-45.900,-179.297,5.693,148.796
C04402=1201.894,44.494,-45.915,-179.295,5.694,148.795
C04403=1201.890,44.743,-45.932,-179.293,5.694,148.795
C04404=1201.884,44.992,-45.948,-179.290,5.695,148.794
C04405=1201.879,45.242,-45.963,-179.288,5.696,148.794
C04406=1201.875,45.491,-45.980,-179.285,5.696,148.793
C04407=1201.869,45.741,-45.995,-179.282,5.698,148.792
C04408=1201.865,45.990,-46.012,-179.279,5.698,148.792
C04409=1201.859,46.240,-46.028,-179.277,5.699,148.791
C04410=1201.854,46.490,-46.044,-179.274,5.700,148.791
C04411=1201.849,46.739,-46.060,-179.272,5.700,148.790
C04412=1201.844,46.988,-46.076,-179.269,5.701,148.789
C04413=1201.840,47.237,-46.092,-179.267,5.702,148.789
C04414=1201.834,47.487,-46.108,-179.264,5.702,148.788
C04415=1201.829,47.737,-46.124,-179.262,5.703,148.787
C04416=1201.824,47.986,-46.140,-179.259,5.703,148.787
C04417=1201.820,48.236,-46.155,-179.257,5.704,148.786
C04418=1201.815,48.484,-46.172,-179.254,5.705,148.786
C04419=1201.810,48.734,-46.188,-179.251,5.706,148.785
C04420=1201.805,48.983,-46.204,-179.248,5.707,148.784
C04421=1201.801,49.233,-46.220,-179.246,5.707,148.784
C04422=1201.795,49.482,-46.237,-179.244,5.708,148.783
C04423=1201.790,49.732,-46.253,-179.241,5.709,148.783
C04424=1201.785,49.981,-46.269,-179.239,5.709,148.782
C04425=1201.780,50.231,-46.285,-179.236,5.710,148.781
C04426=1201.775,50.480,-46.301,-179.234,5.710,148.781
C04427=1201.770,50.730,-46.317,-179.231,5.711,148.780
C04428=1201.765,50.979,-46.334,-179.228,5.713,148.780
C04429=1201.761,51.229,-46.350,-179.226,5.713,148.779
C04430=1201.755,51.478,-46.366,-179.223,5.714,148.778
C04431=1201.751,51.727,-46.382,-179.221,5.715,148.778
C04432=1201.745,51.977,-46.398,-179.218,5.715,148.777
C04433=1201.741,52.226,-46.415,-179.216,5.716,148.777
C04434=1201.736,52.475,-46.431,-179.213,5.716,148.776
C04435=1201.731,52.725,-46.447,-179.211,5.717,148.775
C04436=1201.726,52.974,-46.463,-179.208,5.718,148.775
C04437=1201.721,53.224,-46.479,-179.205,5.719,148.774
C04438=1201.715,53.473,-46.496,-179.202,5.720,148.773
C04439=1201.711,53.723,-46.513,-179.200,5.721,148.773
C04440=1201.705,53.972,-46.528,-179.198,5.721,148.772
C04441=1201.701,54.222,-46.545,-179.195,5.722,148.772
C04442=1201.696,54.470,-46.561,-179.193,5.723,148.771
C04443=1201.691,54.739,-46.579,-179.190,5.724,148.771
C04444=1201.685,55.008,-46.597,-179.187,5.724,148.770
C04445=1201.680,55.277,-46.614,-179.184,5.725,148.769
C04446=1201.675,55.545,-46.632,-179.182,5.726,148.769
C04447=1201.670,55.794,-46.649,-179.178,5.727,148.768
C04448=1201.665,56.044,-46.664,-179.176,5.728,148.767
C04449=1201.660,56.293,-46.682,-179.174,5.728,148.767
C04450=1201.655,56.542,-46.698,-179.171,5.729,148.766
C04451=1201.650,56.792,-46.715,-179.168,5.729,148.765
C04452=1201.645,57.041,-46.730,-179.166,5.730,148.765
C04453=1201.640,57.291,-46.747,-179.164,5.731,148.764
C04454=1201.635,57.540,-46.764,-179.160,5.732,148.764
C04455=1201.630,57.789,-46.781,-179.158,5.733,148.763
C04456=1201.625,58.039,-46.796,-179.156,5.734,148.763
C04457=1201.621,58.289,-46.813,-179.153,5.734,148.762
C04458=1201.616,58.537,-46.829,-179.151,5.735,148.761
C04459=1201.610,58.787,-46.847,-179.148,5.736,148.761
C04460=1201.605,59.036,-46.863,-179.146,5.736,148.760
C04461=1201.601,59.286,-46.880,-179.142,5.738,148.759
C04462=1201.595,59.536,-46.896,-179.140,5.738,148.759
C04463=1201.590,59.785,-46.913,-179.138,5.739,148.758
C04464=1201.586,60.034,-46.929,-179.135,5.740,148.758
C04465=1201.581,60.284,-46.946,-179.133,5.740,148.757
C04466=1201.575,60.533,-46.963,-179.130,5.741,148.757
C04467=1201.571,60.782,-46.979,-179.127,5.742,148.756
C04468=1201.566,61.032,-46.996,-179.125,5.743,148.756
C04469=1201.561,61.281,-47.013,-179.122,5.744,148.755
C04470=1201.556,61.530,-47.030,-179.120,5.744,148.754
C04471=1201.552,61.780,-47.046,-179.117,5.745,148.754
C04472=1201.546,62.029,-47.063,-179.115,5.746,148.753
C04473=1201.541,62.278,-47.080,-179.112,5.747,148.752
C04474=1201.537,62.529,-47.096,-179.109,5.748,148.752
C04475=1201.531,62.778,-47.113,-179.107,5.749,148.751
C04476=1201.526,63.027,-47.129,-179.104,5.749,148.751
C04477=1201.522,63.277,-47.146,-179.102,5.750,148.750
C04478=1201.516,63.526,-47.163,-179.099,5.751,148.750
C04479=1201.512,63.775,-47.180,-179.096,5.752,148.749
C04480=1201.507,64.025,-47.196,-179.094,5.753,148.748
C04481=1201.502,64.274,-47.214,-179.091,5.753,148.748
C04482=1201.497,64.523,-47.231,-179.089,5.754,148.747
C04483=1201.492,64.772,-47.248,-179.086,5.755,148.746
C04484=1201.487,65.022,-47.265,-179.083,5.756,148.746
C04485=1201.482,65.271,-47.281,-179.081,5.757,148.745
C04486=1201.477,65.520,-47.298,-179.078,5.757,148.745
C04487=1201.473,65.770,-47.315,-179.076,5.758,148.744
C04488=1201.467,66.020,-47.332,-179.073,5.759,148.744
C04489=1201.462,66.269,-47.348,-179.071,5.759,148.743
C04490=1201.458,66.518,-47.365,-179.068,5.761,148.743
C04491=1201.453,66.768,-47.382,-179.065,5.762,148.742
C04492=1201.448,67.017,-47.399,-179.063,5.762,148.741
C04493=1201.443,67.266,-47.417,-179.061,5.763,148.741
C04494=1201.438,67.515,-47.433,-179.058,5.764,148.740
C04495=1201.433,67.765,-47.451,-179.055,5.765,148.739
C04496=1201.428,68.015,-47.467,-179.053,5.766,148.739
C04497=1201.423,68.264,-47.484,-179.050,5.767,148.738
C04498=1201.418,68.513,-47.501,-179.047,5.767,148.738
C04499=1201.413,68.762,-47.519,-179.045,5.768,148.737
C04500=1201.409,69.012,-47.535,-179.042,5.769,148.737
C04501=1201.403,69.262,-47.553,-179.039,5.770,148.736
C04502=1201.399,69.511,-47.569,-179.037,5.771,148.736
C04503=1201.393,69.760,-47.586,-179.035,5.771,148.735
C04504=1201.389,70.009,-47.604,-179.032,5.773,148.734
C04505=1201.384,70.259,-47.621,-179.029,5.774,148.734
C04506=1201.379,70.508,-47.638,-179.027,5.774,148.733
C04507=1201.374,70.758,-47.655,-179.024,5.775,148.733
C04508=1201.369,71.006,-47.672,-179.022,5.776,148.732
C04509=1201.364,71.256,-47.689,-179.019,5.777,148.731
C04510=1201.360,71.506,-47.706,-179.016,5.778,148.731
C04511=1201.355,71.755,-47.724,-179.014,5.778,148.730
C04512=1201.350,72.004,-47.741,-179.011,5.779,148.730
C04513=1201.345,72.254,-47.758,-179.009,5.781,148.729
C04514=1201.339,72.503,-47.775,-179.006,5.781,148.729
C04515=1201.335,72.752,-47.792,-179.003,5.782,148.728
C04516=1201.330,73.002,-47.809,-179.001,5.783,148.727
C04517=1201.325,73.252,-47.827,-178.998,5.783,148.727
C04518=1201.320,73.500,-47.844,-178.996,5.785,148.726
C04519=1201.315,73.750,-47.861,-178.993,5.786,148.726
C04520=1201.311,73.999,-47.879,-178.991,5.786,148.725
C04521=1201.305,74.248,-47.895,-178.988,5.787,148.725
C04522=1201.300,74.498,-47.913,-178.985,5.788,148.724
C04523=1201.296,74.747,-47.930,-178.983,5.789,148.723
C04524=1201.291,74.997,-47.947,-178.980,5.790,148.723
C04525=1201.286,75.246,-47.965,-178.978,5.791,148.722
C04526=1201.281,75.495,-47.982,-178.975,5.792,148.722
C04527=1201.276,75.744,-48.000,-178.972,5.793,148.721
C04528=1201.271,75.994,-48.017,-178.970,5.793,148.720
C04529=1201.267,76.244,-48.034,-178.968,5.794,148.720
C04530=1201.262,76.493,-48.052,-178.964,5.796,148.719
C04531=1201.256,76.742,-48.069,-178.962,5.796,148.719
C04532=1201.252,76.991,-48.086,-178.960,5.797,148.718
C04533=1201.246,77.241,-48.103,-178.957,5.798,148.718
C04534=1201.242,77.490,-48.121,-178.954,5.799,148.717
C04535=1201.236,77.740,-48.139,-178.952,5.800,148.717
C04536=1201.232,77.988,-48.156,-178.949,5.801,148.716
C04537=1201.227,78.238,-48.173,-178.947,5.801,148.715
C04538=1201.222,78.487,-48.191,-178.944,5.803,148.715
C04539=1201.217,78.737,-48.209,-178.941,5.803,148.714
C04540=1201.213,78.986,-48.226,-178.939,5.804,148.714
C04541=1201.208,79.235,-48.244,-178.936,5.805,148.713
C04542=1201.203,79.485,-48.261,-178.934,5.807,148.713
C04543=1201.198,79.734,-48.279,-178.931,5.807,148.712
C04544=1201.193,79.984,-48.296,-178.928,5.808,148.711
C04545=1201.188,80.233,-48.314,-178.926,5.809,148.711
C04546=1201.183,80.482,-48.332,-178.923,5.810,148.710
C04547=1201.178,80.751,-48.351,-178.920,5.811,148.710
C04548=1201.172,81.019,-48.370,-178.917,5.812,148.709
C04549=1201.167,81.287,-48.388,-178.915,5.813,148.709
C04550=1201.162,81.556,-48.408,-178.912,5.814,148.708
C04551=1201.157,81.805,-48.424,-178.909,5.815,148.707
C04552=1201.152,82.054,-48.442,-178.907,5.816,148.707
C04553=1201.147,82.303,-48.460,-178.905,5.816,148.706
C04554=1201.142,82.553,-48.478,-178.901,5.818,148.706
C04555=1201.137,82.802,-48.496,-178.899,5.819,148.705
C04556=1201.132,83.052,-48.514,-178.897,5.819,148.704
C04557=1201.128,83.300,-48.531,-178.894,5.821,148.704
C04558=1201.123,83.550,-48.548,-178.891,5.821,148.703
C04559=1201.118,83.799,-48.566,-178.889,5.822,148.703
C04560=1201.113,84.049,-48.584,-178.886,5.823,148.702
C04561=1201.108,84.298,-48.602,-178.883,5.824,148.702
C04562=1201.103,84.548,-48.619,-178.881,5.825,148.701
C04563=1201.098,84.797,-48.637,-178.879,5.826,148.701
C04564=1201.093,85.046,-48.655,-178.876,5.828,148.700
C04565=1201.088,85.295,-48.673,-178.873,5.828,148.700
C04566=1201.083,85.544,-48.691,-178.871,5.829,148.699
C04567=1201.080,85.794,-48.708,-178.868,5.830,148.698
C04568=1201.075,86.044,-48.726,-178.865,5.831,148.698
C04569=1201.070,86.293,-48.744,-178.863,5.832,148.697
C04570=1201.065,86.542,-48.762,-178.860,5.833,148.697
C04571=1201.060,86.791,-48.780,-178.857,5.834,148.696
C04572=1201.055,87.040,-48.798,-178.855,5.835,148.696
C04573=1201.050,87.290,-48.815,-178.853,5.835,148.695
C04574=1201.045,87.539,-48.833,-178.850,5.837,148.695
C04575=1201.040,87.789,-48.851,-178.847,5.838,148.694
C04576=1201.035,88.038,-48.869,-178.845,5.839,148.693
C04577=1201.030,88.287,-48.887,-178.842,5.840,148.693
C04578=1201.026,88.537,-48.906,-178.839,5.841,148.692
C04579=1201.021,88.786,-48.924,-178.837,5.841,148.692
C04580=1201.016,89.035,-48.942,-178.834,5.843,148.691
C04581=1201.011,89.284,-48.960,-178.832,5.844,148.691
C04582=1201.006,89.533,-48.978,-178.829,5.844,148.690
C04583=1201.001,89.783,-48.996,-178.826,5.846,148.690
C04584=1200.996,90.032,-49.014,-178.824,5.847,148.689
C04585=1200.991,90.281,-49.032,-178.821,5.847,148.688
C04586=1200.987,90.531,-49.050,-178.818,5.849,148.688
C04587=1200.982,90.780,-49.068,-178.816,5.850,148.687
C04588=1200.977,91.029,-49.086,-178.814,5.850,148.687
C04589=1200.972,91.278,-49.104,-178.811,5.852,148.686
C04590=1200.967,91.528,-49.122,-178.808,5.853,148.686
C04591=1200.962,91.777,-49.140,-178.806,5.853,148.685
C04592=1200.958,92.027,-49.159,-178.803,5.855,148.685
C04593=1200.953,92.276,-49.177,-178.800,5.856,148.684
C04594=1200.948,92.525,-49.195,-178.798,5.856,148.683
C04595=1200.943,92.774,-49.213,-178.795,5.858,148.683
C04596=1200.938,93.024,-49.231,-178.792,5.859,148.682
C04597=1200.933,93.273,-49.249,-178.790,5.859,148.682
C04598=1200.929,93.523,-49.267,-178.787,5.861,148.681
C04599=1200.924,93.772,-49.285,-178.785,5.862,148.681
C04600=1200.918,94.021,-49.304,-178.782,5.862,148.680
C04601=1200.913,94.271,-49.322,-178.780,5.864,148.680
C04602=1200.909,94.520,-49.341,-178.777,5.865,148.679
C04603=1200.904,94.769,-49.359,-178.774,5.866,148.679
C04604=1200.899,95.018,-49.377,-178.772,5.867,148.678
C04605=1200.894,95.267,-49.395,-178.769,5.868,148.677
C04606=1200.889,95.517,-49.413,-178.766,5.869,148.677
C04607=1200.884,95.767,-49.431,-178.764,5.870,148.676
C04608=1200.880,96.015,-49.450,-178.762,5.871,148.676
C04609=1200.875,96.264,-49.468,-178.758,5.872,148.675
C04610=1200.870,96.514,-49.486,-178.756,5.873,148.675
C04611=1200.865,96.764,-49.505,-178.754,5.874,148.674
C04612=1200.860,97.013,-49.523,-178.751,5.875,148.674
C04613=1200.855,97.261,-49.542,-178.748,5.876,148.673
C04614=1200.851,97.511,-49.560,-178.746,5.878,148.673
C04615=1200.845,97.761,-49.579,-178.743,5.878,148.672
C04616=1200.841,98.009,-49.597,-178.741,5.879,148.672
C04617=1200.836,98.259,-49.615,-178.738,5.881,148.671
C04618=1200.831,98.508,-49.633,-178.736,5.882,148.671
C04619=1200.826,98.758,-49.652,-178.733,5.882,148.670
C04620=1200.821,99.006,-49.671,-178.730,5.884,148.669
C04621=1200.817,99.256,-49.689,-178.728,5.885,148.669
C04622=1200.812,99.506,-49.707,-178.725,5.886,148.668
C04623=1200.807,99.754,-49.727,-178.722,5.887,148.668
C04624=1200.802,100.004,-49.745,-178.720,5.887,148.667
C04625=1200.798,100.253,-49.763,-178.717,5.889,148.667
C04626=1200.792,100.502,-49.782,-178.714,5.890,148.666
C04627=1200.787,100.752,-49.800,-178.712,5.892,148.666
C04628=1200.783,101.000,-49.819,-178.709,5.892,148.665
C04629=1200.778,101.250,-49.838,-178.707,5.893,148.665
C04630=1200.773,101.499,-49.856,-178.704,5.894,148.664
C04631=1200.768,101.748,-49.874,-178.702,5.895,148.664
C04632=1200.763,101.998,-49.893,-178.698,5.897,148.663
C04633=1200.759,102.247,-49.912,-178.696,5.898,148.663
C04634=1200.754,102.497,-49.930,-178.694,5.898,148.662
C04635=1200.749,102.746,-49.949,-178.691,5.900,148.662
C04636=1200.744,102.995,-49.968,-178.688,5.901,148.661
C04637=1200.740,103.245,-49.986,-178.686,5.902,148.661
C04638=1200.734,103.493,-50.005,-178.683,5.903,148.660
C04639=1200.729,103.743,-50.023,-178.681,5.904,148.659
C04640=1200.725,103.992,-50.043,-178.678,5.905,148.659
C04641=1200.720,104.241,-50.061,-178.676,5.906,148.658
C04642=1200.715,104.490,-50.080,-178.672,5.908,148.658
C04643=1200.710,104.740,-50.099,-178.670,5.909,148.657
C04644=1200.705,104.989,-50.117,-178.668,5.909,148.657
C04645=1200.700,105.239,-50.136,-178.665,5.911,148.656
C04646=1200.696,105.487,-50.155,-178.662,5.911,148.656
C04647=1200.690,105.736,-50.174,-178.660,5.913,148.655
C04648=1200.686,105.986,-50.193,-178.657,5.914,148.655
C04649=1200.682,106.235,-50.211,-178.654,5.916,148.654
C04650=1200.677,106.485,-50.230,-178.652,5.916,148.654
C04651=1200.671,106.753,-50.251,-178.649,5.918,148.653
C04652=1200.666,107.021,-50.270,-178.646,5.918,148.653
C04653=1200.661,107.290,-50.291,-178.643,5.920,148.652
C04654=1200.655,107.558,-50.311,-178.641,5.921,148.651
C04655=1200.651,107.808,-50.331,-178.638,5.922,148.651
C04656=1200.646,108.056,-50.350,-178.636,5.923,148.650
C04657=1200.641,108.306,-50.368,-178.633,5.925,148.650
C04658=1200.636,108.555,-50.387,-178.631,5.925,148.649
C04659=1200.632,108.804,-50.406,-178.627,5.927,148.649
C04660=1200.627,109.054,-50.425,-178.625,5.928,148.648
C04661=1200.622,109.302,-50.444,-178.622,5.929,148.648
C04662=1200.617,109.552,-50.463,-178.620,5.930,148.647
C04663=1200.613,109.801,-50.482,-178.617,5.931,148.647
C04664=1200.608,110.051,-50.501,-178.615,5.933,148.646
C04665=1200.602,110.300,-50.520,-178.612,5.933,148.646
C04666=1200.598,110.549,-50.539,-178.609,5.935,148.645
C04667=1200.593,110.798,-50.559,-178.607,5.936,148.645
C04668=1200.589,111.048,-50.577,-178.604,5.937,148.644
C04669=1200.583,111.296,-50.596,-178.602,5.938,148.644
C04670=1200.579,111.546,-50.615,-178.599,5.940,148.643
C04671=1200.574,111.795,-50.635,-178.597,5.940,148.643
C04672=1200.569,112.045,-50.654,-178.593,5.942,148.642
C04673=1200.564,112.293,-50.672,-178.591,5.943,148.642
C04674=1200.559,112.543,-50.692,-178.589,5.943,148.641
C04675=1200.554,112.792,-50.711,-178.586,5.945,148.641
C04676=1200.550,113.041,-50.730,-178.584,5.946,148.640
C04677=1200.545,113.290,-50.750,-178.581,5.948,148.640
C04678=1200.540,113.539,-50.769,-178.578,5.948,148.639
C04679=1200.535,113.789,-50.787,-178.575,5.950,148.639
C04680=1200.530,114.038,-50.807,-178.573,5.951,148.638
C04681=1200.525,114.287,-50.826,-178.570,5.952,148.638
C04682=1200.521,114.536,-50.845,-178.568,5.953,148.637
C04683=1200.516,114.785,-50.865,-178.565,5.955,148.636
C04684=1200.511,115.035,-50.884,-178.563,5.956,148.636
C04685=1200.507,115.284,-50.903,-178.560,5.957,148.636
C04686=1200.502,115.533,-50.923,-178.557,5.958,148.635
C04687=1200.497,115.782,-50.942,-178.555,5.960,148.635
C04688=1200.492,116.031,-50.961,-178.552,5.960,148.634
C04689=1200.487,116.281,-50.981,-178.549,5.962,148.634
C04690=1200.482,116.529,-51.000,-178.547,5.963,148.633
C04691=1200.477,116.779,-51.020,-178.544,5.964,148.633
C04692=1200.473,117.028,-51.039,-178.542,5.965,148.632
C04693=1200.468,117.277,-51.058,-178.539,5.967,148.632
C04694=1200.463,117.527,-51.078,-178.536,5.968,148.631
C04695=1200.458,117.776,-51.097,-178.533,5.969,148.630
C04696=1200.453,118.025,-51.116,-178.531,5.970,148.630
C04697=1200.449,118.274,-51.136,-178.528,5.971,148.629
C04698=1200.444,118.523,-51.155,-178.526,5.972,148.629
C04699=1200.439,118.773,-51.174,-178.523,5.974,148.629
C04700=1200.434,119.022,-51.194,-178.521,5.975,148.628
C04701=1200.429,119.271,-51.213,-178.518,5.976,148.628
C04702=1200.425,119.521,-51.233,-178.515,5.977,148.627
C04703=1200.420,119.769,-51.252,-178.513,5.979,148.627
C04704=1200.415,120.019,-51.271,-178.510,5.980,148.626
C04705=1200.410,120.268,-51.292,-178.507,5.981,148.626
C04706=1200.405,120.517,-51.311,-178.505,5.982,148.625
C04707=1200.400,120.766,-51.331,-178.502,5.984,148.625
C04708=1200.396,121.016,-51.350,-178.500,5.984,148.624
C04709=1200.391,121.264,-51.369,-178.497,5.986,148.624
C04710=1200.386,121.514,-51.389,-178.495,5.987,148.623
C04711=1200.382,121.763,-51.409,-178.492,5.989,148.623
C04712=1200.377,122.012,-51.428,-178.489,5.989,148.622
C04713=1200.372,122.261,-51.448,-178.487,5.991,148.622
C04714=1200.367,122.511,-51.468,-178.484,5.992,148.621
C04715=1200.362,122.760,-51.487,-178.481,5.993,148.621
C04716=1200.358,123.009,-51.507,-178.479,5.994,148.620
C04717=1200.353,123.258,-51.526,-178.476,5.996,148.620
C04718=1200.349,123.508,-51.546,-178.474,5.997,148.619
C04719=1200.343,123.757,-51.565,-178.471,5.998,148.619
C04720=1200.339,124.005,-51.586,-178.468,6.000,148.618
C04721=1200.334,124.255,-51.605,-178.466,6.001,148.618
C04722=1200.329,124.504,-51.625,-178.463,6.002,148.617
C04723=1200.324,124.753,-51.645,-178.461,6.003,148.617
C04724=1200.319,125.002,-51.665,-178.458,6.005,148.616
C04725=1200.315,125.252,-51.684,-178.455,6.005,148.616
C04726=1200.310,125.500,-51.704,-178.453,6.007,148.615
C04727=1200.305,125.750,-51.724,-178.450,6.008,148.615
C04728=1200.300,125.999,-51.744,-178.447,6.010,148.614
C04729=1200.296,126.248,-51.764,-178.445,6.011,148.614
C04730=1200.290,126.497,-51.783,-178.442,6.012,148.613
C04731=1200.286,126.747,-51.803,-178.439,6.014,148.613
C04732=1200.281,126.996,-51.823,-178.437,6.015,148.612
C04733=1200.276,127.245,-51.843,-178.434,6.016,148.612
C04734=1200.272,127.494,-51.863,-178.432,6.017,148.611
C04735=1200.267,127.743,-51.883,-178.429,6.019,148.611
C04736=1200.262,127.993,-51.902,-178.427,6.019,148.610
C04737=1200.258,128.242,-51.923,-178.424,6.021,148.610
C04738=1200.253,128.491,-51.942,-178.421,6.022,148.609
C04739=1200.248,128.739,-51.962,-178.419,6.024,148.609
C04740=1200.243,128.989,-51.982,-178.416,6.025,148.609
C04741=1200.239,129.238,-52.002,-178.413,6.026,148.608
C04742=1200.234,129.488,-52.022,-178.411,6.028,148.608
C04743=1200.229,129.736,-52.042,-178.408,6.029,148.607
C04744=1200.224,129.986,-52.063,-178.405,6.030,148.607
C04745=1200.219,130.235,-52.083,-178.403,6.031,148.606
C04746=1200.214,130.484,-52.102,-178.401,6.033,148.606
C04747=1200.210,130.733,-52.123,-178.397,6.034,148.605
C04748=1200.205,130.983,-52.142,-178.395,6.035,148.605
C04749=1200.201,131.232,-52.163,-178.393,6.037,148.604
C04750=1200.195,131.480,-52.183,-178.390,6.038,148.604
C04751=1200.191,131.729,-52.202,-178.387,6.039,148.603
C04752=1200.186,131.979,-52.223,-178.385,6.041,148.603
C04753=1200.181,132.228,-52.243,-178.382,6.042,148.602
C04754=1200.176,132.477,-52.263,-178.379,6.043,148.602
C04755=1200.171,132.746,-52.285,-178.376,6.045,148.601
C04756=1200.166,133.014,-52.307,-178.374,6.046,148.601
C04757=1200.160,133.283,-52.329,-178.371,6.047,148.600
C04758=1200.156,133.551,-52.350,-178.368,6.049,148.600
C04759=1200.151,133.801,-52.370,-178.365,6.050,148.599
C04760=1200.146,134.050,-52.391,-178.363,6.051,148.599
C04761=1200.141,134.299,-52.411,-178.360,6.053,148.599
C04762=1200.137,134.549,-52.431,-178.358,6.054,148.598
C04763=1200.132,134.797,-52.451,-178.355,6.056,148.597
C04764=1200.127,135.047,-52.472,-178.352,6.057,148.597
C04765=1200.123,135.296,-52.493,-178.350,6.058,148.596
C04766=1200.117,135.545,-52.512,-178.347,6.060,148.596
C04767=1200.113,135.794,-52.532,-178.345,6.061,148.596
C04768=1200.108,136.043,-52.553,-178.342,6.062,148.595
C04769=1200.103,136.292,-52.574,-178.339,6.064,148.595
C04770=1200.099,136.541,-52.593,-178.337,6.065,148.594
C04771=1200.094,136.790,-52.614,-178.334,6.067,148.594
C04772=1200.089,137.040,-52.635,-178.331,6.067,148.593
C04773=1200.085,137.288,-52.655,-178.329,6.069,148.593
C04774=1200.080,137.537,-52.676,-178.326,6.071,148.593
C04775=1200.075,137.787,-52.696,-178.324,6.071,148.592
C04776=1200.070,138.036,-52.716,-178.321,6.073,148.591
C04777=1200.066,138.285,-52.737,-178.318,6.075,148.591
C04778=1200.061,138.534,-52.757,-178.316,6.076,148.590
C04779=1200.056,138.783,-52.778,-178.313,6.077,148.590
C04780=1200.052,139.032,-52.798,-178.311,6.078,148.590
C04781=1200.047,139.282,-52.819,-178.308,6.080,148.589
C04782=1200.042,139.531,-52.840,-178.305,6.081,148.589
C04783=1200.037,139.780,-52.859,-178.303,6.082,148.588
C04784=1200.032,140.029,-52.880,-178.300,6.084,148.588
C04785=1200.028,140.278,-52.901,-178.297,6.086,148.587
C04786=1200.023,140.527,-52.921,-178.295,6.087,148.587
C04787=1200.018,140.777,-52.942,-178.292,6.088,148.587
C04788=1200.014,141.025,-52.962,-178.289,6.090,148.586
C04789=1200.008,141.275,-52.983,-178.287,6.091,148.586
C04790=1200.004,141.524,-53.004,-178.284,6.093,148.585
C04791=1199.999,141.773,-53.025,-178.281,6.094,148.585
C04792=1199.994,142.022,-53.045,-178.279,6.095,148.584
C04793=1199.990,142.271,-53.065,-178.276,6.097,148.584
C04794=1199.985,142.520,-53.086,-178.274,6.098,148.583
C04795=1199.980,142.769,-53.107,-178.271,6.099,148.583
C04796=1199.975,143.018,-53.128,-178.268,6.101,148.582
C04797=1199.971,143.267,-53.148,-178.266,6.102,148.582
C04798=1199.966,143.517,-53.169,-178.263,6.104,148.582
C04799=1199.961,143.765,-53.189,-178.260,6.105,148.581
C04800=1199.956,144.014,-53.211,-178.258,6.106,148.581
C04801=1199.952,144.263,-53.231,-178.255,6.108,148.580
C04802=1199.947,144.512,-53.252,-178.253,6.110,148.580
C04803=1199.942,144.761,-53.273,-178.250,6.110,148.579
C04804=1199.938,145.011,-53.294,-178.248,6.112,148.579
C04805=1199.933,145.260,-53.314,-178.245,6.114,148.578
C04806=1199.928,145.509,-53.335,-178.243,6.115,148.578
C04807=1199.924,145.758,-53.356,-178.240,6.116,148.577
C04808=1199.919,146.007,-53.377,-178.237,6.118,148.577
C04809=1199.914,146.256,-53.398,-178.235,6.119,148.577
C04810=1199.909,146.505,-53.419,-178.232,6.121,148.576
C04811=1199.905,146.754,-53.439,-178.229,6.122,148.576
C04812=1199.900,147.003,-53.460,-178.226,6.124,148.575
C04813=1199.895,147.252,-53.481,-178.224,6.125,148.575
C04814=1199.891,147.502,-53.503,-178.221,6.127,148.574
C04815=1199.886,147.751,-53.524,-178.218,6.128,148.574
C04816=1199.881,148.000,-53.544,-178.216,6.129,148.573
C04817=1199.876,148.249,-53.565,-178.213,6.131,148.573
C04818=1199.872,148.498,-53.586,-178.211,6.133,148.573
C04819=1199.867,148.747,-53.607,-178.208,6.133,148.572
C04820=1199.862,148.996,-53.628,-178.206,6.135,148.572
C04821=1199.858,149.245,-53.649,-178.203,6.137,148.571
C04822=1199.853,149.494,-53.670,-178.201,6.138,148.571
C04823=1199.848,149.744,-53.691,-178.198,6.139,148.570
C04824=1199.844,149.992,-53.712,-178.195,6.141,148.570
C04825=1199.838,150.241,-53.733,-178.192,6.143,148.570
C04826=1199.833,150.490,-53.754,-178.190,6.144,148.569
C04827=1199.830,150.739,-53.776,-178.187,6.145,148.569
C04828=1199.824,150.989,-53.797,-178.184,6.147,148.568
C04829=1199.819,151.238,-53.818,-178.182,6.148,148.568
C04830=1199.815,151.486,-53.839,-178.179,6.150,148.567
C04831=1199.810,151.736,-53.860,-178.177,6.151,148.567
C04832=1199.806,151.985,-53.882,-178.174,6.153,148.566
C04833=1199.801,152.234,-53.903,-178.172,6.154,148.566
C04834=1199.796,152.483,-53.923,-178.169,6.156,148.566
C04835=1199.791,152.732,-53.945,-178.166,6.157,148.565
C04836=1199.786,152.981,-53.966,-178.164,6.158,148.565
C04837=1199.783,153.230,-53.987,-178.161,6.160,148.564
C04838=1199.777,153.479,-54.008,-178.158,6.162,148.564
C04839=1199.773,153.728,-54.030,-178.156,6.163,148.564
C04840=1199.767,153.977,-54.051,-178.153,6.164,148.563
C04841=1199.763,154.227,-54.073,-178.150,6.166,148.563
C04842=1199.759,154.476,-54.093,-178.148,6.168,148.562
C04843=1199.754,154.724,-54.115,-178.145,6.169,148.562
C04844=1199.749,154.973,-54.136,-178.143,6.170,148.561
C04845=1199.744,155.223,-54.158,-178.140,6.172,148.561
C04846=1199.739,155.472,-54.179,-178.137,6.174,148.560
C04847=1199.735,155.720,-54.200,-178.135,6.175,148.560
C04848=1199.730,155.969,-54.222,-178.132,6.176,148.560
C04849=1199.726,156.219,-54.243,-178.130,6.178,148.559
C04850=1199.721,156.468,-54.265,-178.127,6.180,148.559
C04851=1199.716,156.717,-54.286,-178.124,6.181,148.558
C04852=1199.711,156.966,-54.308,-178.122,6.182,148.558
C04853=1199.707,157.215,-54.329,-178.119,6.184,148.558
C04854=1199.702,157.464,-54.350,-178.116,6.186,148.557
C04855=1199.697,157.712,-54.371,-178.114,6.187,148.557
C04856=1199.693,157.962,-54.394,-178.111,6.189,148.556
C04857=1199.688,158.211,-54.414,-178.108,6.190,148.556
C04858=1199.683,158.460,-54.436,-178.106,6.192,148.555
C04859=1199.678,158.729,-54.459,-178.103,6.194,148.555
C04860=1199.673,158.998,-54.482,-178.100,6.195,148.555
C04861=1199.668,159.266,-54.506,-178.097,6.197,148.554
C04862=1199.663,159.536,-54.529,-178.094,6.199,148.554
C04863=1199.658,159.785,-54.551,-178.092,6.200,148.553
C04864=1199.653,160.034,-54.573,-178.089,6.201,148.553
C04865=1199.648,160.283,-54.594,-178.086,6.203,148.552
C04866=1199.644,160.532,-54.616,-178.084,6.205,148.552
C04867=1199.639,160.781,-54.638,-178.081,6.206,148.552
C04868=1199.634,161.030,-54.659,-178.079,6.207,148.551
C04869=1199.630,161.280,-54.681,-178.076,6.209,148.551
C04870=1199.625,161.528,-54.702,-178.073,6.211,148.550
C04871=1199.621,161.778,-54.724,-178.071,6.212,148.550
C04872=1199.616,162.026,-54.746,-178.068,6.213,148.550
C04873=1199.611,162.275,-54.768,-178.066,6.215,148.549
C04874=1199.607,162.524,-54.790,-178.063,6.217,148.549
C04875=1199.601,162.774,-54.811,-178.060,6.219,148.548
C04876=1199.597,163.023,-54.833,-178.058,6.221,148.548
C04877=1199.592,163.272,-54.854,-178.055,6.221,148.547
C04878=1199.587,163.520,-54.876,-178.052,6.223,148.547
C04879=1199.583,163.770,-54.898,-178.050,6.225,148.547
C04880=1199.578,164.018,-54.920,-178.047,6.227,148.546
C04881=1199.574,164.267,-54.942,-178.044,6.228,148.546
C04882=1199.569,164.516,-54.964,-178.042,6.229,148.546
C04883=1199.564,164.765,-54.985,-178.040,6.231,148.545
C04884=1199.560,165.014,-55.007,-178.037,6.233,148.545
C04885=1199.555,165.263,-55.029,-178.034,6.234,148.544
C04886=1199.551,165.512,-55.051,-178.031,6.236,148.544
C04887=1199.546,165.761,-55.073,-178.029,6.237,148.544
C04888=1199.542,166.010,-55.095,-178.026,6.239,148.543
C04889=1199.537,166.259,-55.116,-178.024,6.241,148.543
C04890=1199.532,166.508,-55.139,-178.021,6.243,148.542
C04891=1199.527,166.757,-55.161,-178.018,6.244,148.542
C04892=1199.523,167.006,-55.183,-178.016,6.245,148.541
C04893=1199.518,167.255,-55.204,-178.013,6.247,148.541
C04894=1199.514,167.504,-55.227,-178.010,6.249,148.541
C04895=1199.509,167.753,-55.248,-178.008,6.250,148.540
C04896=1199.504,168.002,-55.270,-178.005,6.252,148.540
C04897=1199.499,168.251,-55.293,-178.002,6.254,148.540
C04898=1199.495,168.501,-55.315,-178.000,6.255,148.539
C04899=1199.490,168.749,-55.336,-177.998,6.257,148.539
C04900=1199.485,168.999,-55.358,-177.995,6.258,148.538
C04901=1199.481,169.247,-55.381,-177.992,6.260,148.538
C04902=1199.476,169.496,-55.403,-177.989,6.262,148.538
C04903=1199.471,169.745,-55.425,-177.987,6.264,148.537
C04904=1199.467,169.994,-55.447,-177.984,6.265,148.537
C04905=1199.462,170.243,-55.469,-177.982,6.266,148.536
C04906=1199.457,170.493,-55.491,-177.979,6.268,148.536
C04907=1199.452,170.741,-55.514,-177.976,6.270,148.536
C04908=1199.448,170.990,-55.536,-177.974,6.272,148.535
C04909=1199.443,171.239,-55.558,-177.971,6.274,148.535
C04910=1199.438,171.488,-55.580,-177.969,6.274,148.534
C04911=1199.434,171.736,-55.603,-177.966,6.276,148.534
C04912=1199.429,171.986,-55.625,-177.963,6.278,148.534
C04913=1199.425,172.235,-55.647,-177.960,6.280,148.533
C04914=1199.419,172.484,-55.669,-177.958,6.281,148.533
C04915=1199.415,172.733,-55.692,-177.955,6.283,148.533
C04916=1199.411,172.981,-55.713,-177.952,6.285,148.532
C04917=1199.406,173.231,-55.736,-177.950,6.286,148.532
C04918=1199.402,173.480,-55.759,-177.948,6.288,148.531
C04919=1199.397,173.728,-55.780,-177.945,6.290,148.531
C04920=1199.392,173.978,-55.803,-177.942,6.291,148.531
C04921=1199.387,174.226,-55.826,-177.939,6.293,148.530
C04922=1199.383,174.475,-55.848,-177.937,6.295,148.530
C04923=1199.378,174.725,-55.870,-177.934,6.296,148.529
C04924=1199.373,174.973,-55.893,-177.932,6.297,148.529
C04925=1199.369,175.222,-55.915,-177.929,6.299,148.529
C04926=1199.363,175.471,-55.937,-177.926,6.301,148.528
C04927=1199.360,175.720,-55.960,-177.924,6.303,148.528
C04928=1199.355,175.970,-55.982,-177.921,6.305,148.528
C04929=1199.350,176.218,-56.005,-177.918,6.306,148.527
C04930=1199.346,176.467,-56.027,-177.916,6.308,148.527
C04931=1199.341,176.716,-56.050,-177.913,6.310,148.527
C04932=1199.336,176.965,-56.072,-177.911,6.311,148.526
C04933=1199.331,177.214,-56.095,-177.908,6.313,148.526
C04934=1199.327,177.463,-56.117,-177.906,6.315,148.525
C04935=1199.322,177.711,-56.140,-177.903,6.316,148.525
C04936=1199.318,177.961,-56.162,-177.900,6.318,148.525
C04937=1199.314,178.209,-56.185,-177.898,6.320,148.524
C04938=1199.308,178.458,-56.207,-177.895,6.321,148.524
C04939=1199.304,178.707,-56.230,-177.892,6.323,148.523
C04940=1199.299,178.957,-56.253,-177.889,6.325,148.523
C04941=1199.294,179.205,-56.275,-177.887,6.326,148.523
C04942=1199.289,179.454,-56.298,-177.884,6.328,148.522
C04943=1199.286,179.703,-56.321,-177.882,6.330,148.522
C04944=1199.281,179.952,-56.344,-177.879,6.331,148.522
C04945=1199.276,180.201,-56.366,-177.876,6.333,148.521
C04946=1199.271,180.450,-56.389,-177.874,6.335,148.521
C04947=1199.267,180.699,-56.411,-177.871,6.337,148.521
C04948=1199.262,180.947,-56.434,-177.869,6.339,148.520
C04949=1199.257,181.196,-56.457,-177.866,6.340,148.520
C04950=1199.253,181.446,-56.479,-177.863,6.342,148.519
C04951=1199.248,181.695,-56.503,-177.861,6.344,148.519
C04952=1199.243,181.943,-56.525,-177.858,6.345,148.519
C04953=1199.238,182.193,-56.548,-177.856,6.347,148.518
C04954=1199.234,182.441,-56.571,-177.853,6.349,148.518
C04955=1199.230,182.690,-56.594,-177.850,6.350,148.518
C04956=1199.224,182.939,-56.617,-177.848,6.352,148.517
C04957=1199.220,183.188,-56.639,-177.845,6.354,148.517
C04958=1199.215,183.437,-56.662,-177.842,6.356,148.517
C04959=1199.212,183.686,-56.685,-177.840,6.358,148.516
C04960=1199.207,183.935,-56.708,-177.837,6.359,148.516
C04961=1199.201,184.184,-56.731,-177.834,6.361,148.516
C04962=1199.197,184.432,-56.753,-177.832,6.363,148.515
C04963=1199.192,184.702,-56.779,-177.829,6.365,148.515
C04964=1199.187,184.972,-56.803,-177.826,6.366,148.514
C04965=1199.182,185.241,-56.828,-177.823,6.368,148.514
C04966=1199.177,185.511,-56.854,-177.821,6.370,148.514
C04967=1199.173,185.760,-56.876,-177.818,6.372,148.513
C04968=1199.168,186.009,-56.899,-177.815,6.374,148.513
C04969=1199.163,186.258,-56.923,-177.813,6.375,148.512
C04970=1199.159,186.506,-56.945,-177.810,6.377,148.512
C04971=1199.154,186.755,-56.968,-177.807,6.379,148.512
C04972=1199.149,187.004,-56.992,-177.805,6.381,148.511
C04973=1199.145,187.253,-57.015,-177.802,6.383,148.511
C04974=1199.141,187.502,-57.038,-177.799,6.384,148.511
C04975=1199.136,187.751,-57.061,-177.797,6.386,148.510
C04976=1199.131,188.000,-57.084,-177.794,6.388,148.510
C04977=1199.126,188.248,-57.107,-177.791,6.390,148.510
C04978=1199.122,188.498,-57.130,-177.789,6.392,148.509
C04979=1199.117,188.747,-57.153,-177.786,6.393,148.509
C04980=1199.112,188.996,-57.176,-177.783,6.395,148.509
C04981=1199.108,189.245,-57.200,-177.781,6.397,148.508
C04982=1199.103,189.494,-57.223,-177.778,6.399,148.508
C04983=1199.099,189.742,-57.246,-177.775,6.401,148.508
C04984=1199.095,189.991,-57.270,-177.773,6.403,148.507
C04985=1199.089,190.239,-57.293,-177.770,6.404,148.507
C04986=1199.085,190.488,-57.316,-177.767,6.406,148.506
C04987=1199.080,190.737,-57.339,-177.765,6.408,148.506
C04988=1199.076,190.986,-57.362,-177.763,6.410,148.506
C04989=1199.071,191.235,-57.386,-177.761,6.411,148.506
C04990=1199.067,191.484,-57.409,-177.758,6.413,148.505
C04991=1199.062,191.733,-57.432,-177.755,6.415,148.505
C04992=1199.057,191.982,-57.456,-177.753,6.416,148.505
C04993=1199.052,192.231,-57.479,-177.750,6.418,148.504
C04994=1199.048,192.480,-57.502,-177.747,6.420,148.504
C04995=1199.043,192.729,-57.526,-177.745,6.422,148.504
C04996=1199.039,192.977,-57.549,-177.742,6.424,148.503
C04997=1199.035,193.226,-57.573,-177.739,6.426,148.503
C04998=1199.030,193.475,-57.596,-177.737,6.427,148.502
C04999=1199.025,193.724,-57.619,-177.734,6.429,148.502
C05000=1199.021,193.973,-57.643,-177.731,6.431,148.502
C05001=1199.016,194.221,-57.666,-177.729,6.433,148.501
C05002=1199.011,194.470,-57.690,-177.726,6.435,148.501
C05003=1199.006,194.719,-57.713,-177.723,6.436,148.501
C05004=1199.002,194.968,-57.737,-177.721,6.438,148.500
C05005=1198.997,195.217,-57.761,-177.718,6.440,148.500
C05006=1198.992,195.466,-57.784,-177.716,6.442,148.500
C05007=1198.988,195.715,-57.807,-177.713,6.444,148.500
C05008=1198.983,195.963,-57.831,-177.711,6.446,148.499
C05009=1198.979,196.212,-57.855,-177.708,6.448,148.499
C05010=1198.974,196.461,-57.878,-177.705,6.449,148.499
C05011=1198.970,196.710,-57.902,-177.703,6.451,148.498
C05012=1198.965,196.959,-57.925,-177.700,6.453,148.498
C05013=1198.961,197.208,-57.949,-177.697,6.455,148.497
C05014=1198.956,197.457,-57.973,-177.695,6.457,148.497
C05015=1198.952,197.706,-57.997,-177.691,6.459,148.497
C05016=1198.947,197.955,-58.020,-177.689,6.461,148.496
C05017=1198.943,198.203,-58.044,-177.686,6.463,148.496
C05018=1198.938,198.452,-58.067,-177.683,6.465,148.496
C05019=1198.933,198.701,-58.092,-177.681,6.467,148.496
C05020=1198.929,198.950,-58.115,-177.679,6.469,148.495
C05021=1198.924,199.198,-58.139,-177.676,6.471,148.495
C05022=1198.920,199.447,-58.162,-177.673,6.472,148.495
C05023=1198.915,199.696,-58.186,-177.671,6.474,148.494
C05024=1198.910,199.945,-58.210,-177.668,6.476,148.494
C05025=1198.905,200.193,-58.234,-177.665,6.478,148.494
C05026=1198.901,200.442,-58.258,-177.663,6.480,148.493
C05027=1198.896,200.691,-58.282,-177.660,6.481,148.493
C05028=1198.892,200.940,-58.306,-177.657,6.483,148.493
C05029=1198.888,201.189,-58.330,-177.655,6.485,148.492
C05030=1198.883,201.438,-58.353,-177.653,6.487,148.492
C05031=1198.879,201.686,-58.377,-177.650,6.489,148.492
C05032=1198.873,201.936,-58.401,-177.647,6.491,148.491
C05033=1198.869,202.184,-58.425,-177.645,6.493,148.491
C05034=1198.864,202.433,-58.448,-177.642,6.495,148.491
C05035=1198.860,202.682,-58.473,-177.639,6.496,148.490
C05036=1198.856,202.931,-58.497,-177.637,6.498,148.490
C05037=1198.851,203.180,-58.521,-177.634,6.500,148.490
C05038=1198.846,203.428,-58.545,-177.632,6.502,148.490
C05039=1198.842,203.677,-58.569,-177.629,6.505,148.489
C05040=1198.837,203.926,-58.592,-177.626,6.507,148.489
C05041=1198.833,204.174,-58.617,-177.623,6.508,148.489
C05042=1198.828,204.423,-58.641,-177.621,6.510,148.488
C05043=1198.823,204.673,-58.665,-177.618,6.512,148.488
C05044=1198.819,204.921,-58.689,-177.615,6.514,148.488
C05045=1198.815,205.170,-58.713,-177.613,6.516,148.487
C05046=1198.809,205.419,-58.737,-177.610,6.518,148.487
C05047=1198.805,205.667,-58.761,-177.608,6.520,148.487
C05048=1198.801,205.916,-58.786,-177.605,6.521,148.486
C05049=1198.797,206.165,-58.810,-177.603,6.523,148.486
C05050=1198.791,206.414,-58.834,-177.600,6.525,148.486
C05051=1198.787,206.663,-58.858,-177.597,6.527,148.485
C05052=1198.782,206.911,-58.882,-177.594,6.530,148.485
C05053=1198.778,207.160,-58.907,-177.592,6.532,148.485
C05054=1198.774,207.409,-58.931,-177.589,6.534,148.485
C05055=1198.769,207.658,-58.954,-177.587,6.535,148.484
C05056=1198.764,207.907,-58.979,-177.584,6.537,148.484
C05057=1198.759,208.155,-59.003,-177.581,6.539,148.484
C05058=1198.756,208.404,-59.027,-177.579,6.541,148.483
C05059=1198.750,208.653,-59.052,-177.576,6.543,148.483
C05060=1198.746,208.901,-59.076,-177.574,6.545,148.483
C05061=1198.741,209.150,-59.101,-177.571,6.547,148.482
C05062=1198.737,209.399,-59.125,-177.568,6.548,148.482
C05063=1198.732,209.648,-59.149,-177.565,6.551,148.482
C05064=1198.727,209.897,-59.173,-177.563,6.553,148.481
C05065=1198.723,210.145,-59.197,-177.560,6.555,148.481
C05066=1198.718,210.395,-59.222,-177.558,6.557,148.481
C05067=1198.714,210.665,-59.248,-177.555,6.559,148.481
C05068=1198.709,210.935,-59.275,-177.552,6.561,148.480
C05069=1198.704,211.205,-59.302,-177.549,6.563,148.480
C05070=1198.699,211.476,-59.328,-177.547,6.565,148.480
C05071=1198.694,211.725,-59.352,-177.543,6.568,148.479
C05072=1198.689,211.973,-59.377,-177.541,6.569,148.479
C05073=1198.685,212.223,-59.401,-177.538,6.571,148.479
C05074=1198.681,212.471,-59.427,-177.536,6.573,148.479
C05075=1198.676,212.719,-59.451,-177.533,6.575,148.478
C05076=1198.672,212.969,-59.476,-177.531,6.577,148.478
C05077=1198.667,213.217,-59.500,-177.528,6.579,148.478
C05078=1198.662,213.466,-59.525,-177.525,6.581,148.477
C05079=1198.658,213.715,-59.549,-177.523,6.584,148.477
C05080=1198.653,213.964,-59.574,-177.520,6.586,148.477
C05081=1198.649,214.212,-59.598,-177.517,6.587,148.477
C05082=1198.644,214.461,-59.623,-177.515,6.589,148.476
C05083=1198.639,214.710,-59.648,-177.512,6.591,148.476
C05084=1198.635,214.958,-59.672,-177.510,6.593,148.476
C05085=1198.631,215.207,-59.697,-177.507,6.595,148.475
C05086=1198.626,215.456,-59.721,-177.504,6.598,148.475
C05087=1198.621,215.704,-59.746,-177.501,6.599,148.475
C05088=1198.617,215.954,-59.771,-177.499,6.601,148.474
C05089=1198.612,216.202,-59.796,-177.497,6.603,148.474
C05090=1198.608,216.451,-59.821,-177.494,6.605,148.474
C05091=1198.603,216.699,-59.845,-177.491,6.607,148.474
C05092=1198.598,216.948,-59.870,-177.489,6.609,148.473
C05093=1198.595,217.197,-59.895,-177.485,6.612,148.473
C05094=1198.590,217.445,-59.920,-177.483,6.614,148.473
C05095=1198.585,217.695,-59.945,-177.481,6.616,148.473
C05096=1198.581,217.943,-59.969,-177.478,6.617,148.472
C05097=1198.576,218.191,-59.994,-177.475,6.619,148.472
C05098=1198.571,218.441,-60.019,-177.473,6.621,148.472
C05099=1198.567,218.689,-60.043,-177.470,6.624,148.471
C05100=1198.563,218.938,-60.069,-177.467,6.626,148.471
C05101=1198.558,219.187,-60.094,-177.465,6.628,148.471
C05102=1198.554,219.436,-60.118,-177.462,6.630,148.471
C05103=1198.549,219.684,-60.143,-177.460,6.632,148.470
C05104=1198.545,219.933,-60.168,-177.457,6.633,148.470
C05105=1198.540,220.181,-60.193,-177.455,6.635,148.470
C05106=1198.536,220.431,-60.218,-177.452,6.638,148.470
C05107=1198.531,220.679,-60.243,-177.449,6.640,148.469
C05108=1198.526,220.927,-60.268,-177.447,6.642,148.469
C05109=1198.522,221.177,-60.293,-177.444,6.644,148.469
C05110=1198.517,221.425,-60.318,-177.442,6.646,148.469
C05111=1198.513,221.674,-60.343,-177.439,6.648,148.468
C05112=1198.508,221.922,-60.369,-177.436,6.650,148.468
C05113=1198.504,222.171,-60.393,-177.433,6.652,148.468
C05114=1198.499,222.419,-60.418,-177.431,6.654,148.467
C05115=1198.495,222.669,-60.443,-177.428,6.656,148.467
C05116=1198.490,222.917,-60.469,-177.426,6.658,148.467
C05117=1198.485,223.166,-60.494,-177.423,6.661,148.467
C05118=1198.482,223.415,-60.519,-177.420,6.663,148.466
C05119=1198.477,223.664,-60.544,-177.418,6.665,148.466
C05120=1198.473,223.912,-60.569,-177.415,6.667,148.466
C05121=1198.468,224.160,-60.595,-177.413,6.669,148.466
C05122=1198.463,224.410,-60.620,-177.410,6.671,148.465
C05123=1198.458,224.658,-60.645,-177.407,6.673,148.465
C05124=1198.455,224.907,-60.670,-177.404,6.675,148.465
C05125=1198.450,225.155,-60.695,-177.402,6.677,148.465
C05126=1198.446,225.404,-60.721,-177.400,6.679,148.464
C05127=1198.440,225.653,-60.745,-177.397,6.681,148.464
C05128=1198.436,225.902,-60.771,-177.394,6.684,148.464
C05129=1198.432,226.150,-60.797,-177.392,6.686,148.464
C05130=1198.427,226.399,-60.822,-177.389,6.687,148.463
C05131=1198.423,226.648,-60.847,-177.387,6.690,148.463
C05132=1198.418,226.896,-60.873,-177.384,6.691,148.463
C05133=1198.413,227.145,-60.898,-177.381,6.694,148.462
C05134=1198.409,227.394,-60.924,-177.378,6.696,148.462
C05135=1198.405,227.642,-60.948,-177.376,6.698,148.462
C05136=1198.401,227.891,-60.974,-177.374,6.700,148.462
C05137=1198.396,228.140,-60.999,-177.371,6.702,148.461
C05138=1198.391,228.388,-61.025,-177.368,6.705,148.461
C05139=1198.387,228.637,-61.050,-177.366,6.707,148.461
C05140=1198.382,228.885,-61.076,-177.363,6.708,148.461
C05141=1198.378,229.134,-61.101,-177.361,6.711,148.461
C05142=1198.373,229.383,-61.126,-177.358,6.713,148.460
C05143=1198.369,229.632,-61.152,-177.355,6.715,148.460
C05144=1198.365,229.880,-61.178,-177.353,6.717,148.460
C05145=1198.360,230.128,-61.203,-177.350,6.719,148.460
C05146=1198.356,230.377,-61.229,-177.347,6.721,148.459
C05147=1198.351,230.626,-61.254,-177.345,6.724,148.459
C05148=1198.346,230.874,-61.280,-177.342,6.726,148.459
C05149=1198.341,231.123,-61.306,-177.339,6.728,148.458
C05150=1198.337,231.373,-61.331,-177.337,6.730,148.458
C05151=1198.332,231.621,-61.357,-177.334,6.732,148.458
C05152=1198.328,231.870,-61.382,-177.331,6.734,148.458
C05153=1198.324,232.118,-61.408,-177.329,6.736,148.458
C05154=1198.319,232.367,-61.434,-177.327,6.738,148.457
C05155=1198.315,232.615,-61.459,-177.325,6.740,148.457
C05156=1198.310,232.864,-61.485,-177.321,6.743,148.457
C05157=1198.306,233.113,-61.511,-177.319,6.745,148.457
C05158=1198.301,233.361,-61.536,-177.317,6.747,148.456
C05159=1198.297,233.610,-61.562,-177.314,6.749,148.456
C05160=1198.292,233.859,-61.588,-177.311,6.752,148.456
C05161=1198.287,234.107,-61.614,-177.309,6.754,148.456
C05162=1198.283,234.356,-61.639,-177.306,6.756,148.455
C05163=1198.279,234.605,-61.665,-177.304,6.758,148.455
C05164=1198.275,234.854,-61.691,-177.301,6.760,148.455
C05165=1198.270,235.101,-61.717,-177.298,6.762,148.455
C05166=1198.265,235.350,-61.743,-177.296,6.764,148.455
C05167=1198.261,235.599,-61.769,-177.293,6.766,148.454
C05168=1198.257,235.848,-61.795,-177.290,6.769,148.454
C05169=1198.252,236.096,-61.820,-177.288,6.771,148.454
C05170=1198.248,236.345,-61.846,-177.285,6.773,148.454
C05171=1198.243,236.616,-61.875,-177.282,6.776,148.454
C05172=1198.238,236.888,-61.903,-177.280,6.778,148.453
C05173=1198.233,237.159,-61.931,-177.277,6.780,148.453
C05174=1198.228,237.431,-61.960,-177.274,6.782,148.453
C05175=1198.224,237.679,-61.986,-177.271,6.785,148.453
C05176=1198.219,237.929,-62.012,-177.269,6.787,148.452
C05177=1198.214,238.176,-62.038,-177.266,6.789,148.452
C05178=1198.210,238.425,-62.064,-177.264,6.791,148.452
C05179=1198.206,238.674,-62.089,-177.261,6.794,148.452
C05180=1198.201,238.923,-62.116,-177.258,6.796,148.451
C05181=1198.197,239.171,-62.142,-177.256,6.798,148.451
C05182=1198.192,239.419,-62.168,-177.253,6.801,148.451
C05183=1198.187,239.668,-62.194,-177.250,6.803,148.451
C05184=1198.183,239.917,-62.220,-177.248,6.804,148.450
C05185=1198.179,240.165,-62.246,-177.246,6.807,148.450
C05186=1198.174,240.414,-62.273,-177.242,6.809,148.450
C05187=1198.170,240.662,-62.299,-177.240,6.811,148.450
C05188=1198.166,240.911,-62.324,-177.238,6.813,148.450
C05189=1198.161,241.160,-62.351,-177.235,6.816,148.450
C05190=1198.157,241.408,-62.377,-177.232,6.818,148.449
C05191=1198.152,241.657,-62.403,-177.230,6.820,148.449
C05192=1198.147,241.906,-62.429,-177.227,6.822,148.449
C05193=1198.144,242.154,-62.456,-177.224,6.825,148.449
C05194=1198.139,242.403,-62.482,-177.222,6.827,148.448
C05195=1198.135,242.651,-62.509,-177.219,6.829,148.448
C05196=1198.129,242.900,-62.535,-177.217,6.832,148.448
C05197=1198.125,243.148,-62.561,-177.214,6.834,148.448
C05198=1198.121,243.397,-62.587,-177.212,6.836,148.448
C05199=1198.116,243.645,-62.614,-177.209,6.838,148.447
C05200=1198.112,243.894,-62.640,-177.207,6.841,148.447
C05201=1198.107,244.142,-62.667,-177.204,6.842,148.447
C05202=1198.103,244.391,-62.692,-177.202,6.845,148.447
C05203=1198.099,244.640,-62.720,-177.199,6.847,148.447
C05204=1198.094,244.889,-62.745,-177.196,6.849,148.446
C05205=1198.090,245.137,-62.772,-177.194,6.851,148.446
C05206=1198.085,245.386,-62.798,-177.191,6.854,148.446
C05207=1198.081,245.634,-62.825,-177.189,6.856,148.446
C05208=1198.077,245.883,-62.852,-177.186,6.858,148.446
C05209=1198.071,246.131,-62.878,-177.183,6.861,148.445
C05210=1198.067,246.379,-62.904,-177.181,6.863,148.445
C05211=1198.062,246.628,-62.930,-177.178,6.865,148.445
C05212=1198.058,246.876,-62.957,-177.175,6.868,148.445
C05213=1198.054,247.125,-62.984,-177.173,6.870,148.445
C05214=1198.050,247.374,-63.010,-177.170,6.872,148.444
C05215=1198.045,247.622,-63.037,-177.168,6.875,148.444
C05216=1198.041,247.870,-63.063,-177.165,6.876,148.444
C05217=1198.036,248.119,-63.090,-177.163,6.879,148.444
C05218=1198.031,248.368,-63.117,-177.160,6.881,148.444
C05219=1198.027,248.616,-63.143,-177.158,6.883,148.444
C05220=1198.023,248.865,-63.170,-177.155,6.885,148.443
C05221=1198.019,249.113,-63.196,-177.152,6.888,148.443
C05222=1198.014,249.362,-63.223,-177.150,6.890,148.443
C05223=1198.009,249.610,-63.250,-177.147,6.892,148.443
C05224=1198.005,249.859,-63.276,-177.144,6.895,148.442
C05225=1198.001,250.107,-63.304,-177.142,6.897,148.442
C05226=1197.996,250.356,-63.330,-177.139,6.899,148.442
C05227=1197.992,250.604,-63.356,-177.137,6.902,148.442
C05228=1197.987,250.853,-63.383,-177.135,6.904,148.442
C05229=1197.983,251.102,-63.411,-177.131,6.907,148.442
C05230=1197.979,251.350,-63.437,-177.129,6.909,148.442
C05231=1197.975,251.599,-63.464,-177.127,6.911,148.441
C05232=1197.970,251.847,-63.491,-177.124,6.914,148.441
C05233=1197.966,252.096,-63.517,-177.121,6.916,148.441
C05234=1197.961,252.345,-63.544,-177.119,6.918,148.441
C05235=1197.956,252.593,-63.571,-177.116,6.921,148.441
C05236=1197.952,252.842,-63.598,-177.114,6.923,148.440
C05237=1197.948,253.090,-63.625,-177.111,6.925,148.440
C05238=1197.943,253.338,-63.652,-177.108,6.928,148.440
C05239=1197.938,253.587,-63.679,-177.106,6.930,148.440
C05240=1197.934,253.835,-63.706,-177.103,6.932,148.440
C05241=1197.930,254.084,-63.733,-177.101,6.935,148.440
C05242=1197.926,254.333,-63.760,-177.098,6.936,148.439
C05243=1197.921,254.581,-63.787,-177.096,6.939,148.439
C05244=1197.917,254.830,-63.814,-177.093,6.941,148.439
C05245=1197.913,255.078,-63.841,-177.090,6.944,148.439
C05246=1197.908,255.326,-63.868,-177.088,6.946,148.439
C05247=1197.903,255.575,-63.895,-177.085,6.948,148.438
C05248=1197.899,255.823,-63.922,-177.083,6.951,148.438
C05249=1197.895,256.073,-63.949,-177.080,6.953,148.438
C05250=1197.890,256.321,-63.976,-177.078,6.955,148.438
C05251=1197.886,256.569,-64.003,-177.075,6.958,148.438
C05252=1197.882,256.817,-64.030,-177.073,6.960,148.438
C05253=1197.877,257.066,-64.057,-177.070,6.963,148.438
C05254=1197.872,257.314,-64.085,-177.067,6.965,148.437
C05255=1197.868,257.563,-64.112,-177.065,6.967,148.437
C05256=1197.864,257.812,-64.139,-177.062,6.970,148.437
C05257=1197.859,258.060,-64.166,-177.060,6.972,148.437
C05258=1197.855,258.308,-64.194,-177.057,6.975,148.437
C05259=1197.851,258.556,-64.220,-177.054,6.977,148.437
C05260=1197.846,258.805,-64.247,-177.052,6.980,148.436
C05261=1197.842,259.054,-64.275,-177.049,6.982,148.436
C05262=1197.838,259.302,-64.303,-177.047,6.984,148.436
C05263=1197.833,259.550,-64.330,-177.044,6.987,148.436
C05264=1197.828,259.799,-64.357,-177.042,6.989,148.436
C05265=1197.824,260.048,-64.384,-177.039,6.992,148.436
C05266=1197.820,260.296,-64.412,-177.036,6.994,148.435
C05267=1197.815,260.544,-64.439,-177.034,6.996,148.435
C05268=1197.811,260.793,-64.466,-177.031,6.999,148.435
C05269=1197.806,261.041,-64.494,-177.029,7.001,148.435
C05270=1197.802,261.290,-64.521,-177.026,7.004,148.435
C05271=1197.798,261.539,-64.548,-177.023,7.005,148.435
C05272=1197.793,261.786,-64.576,-177.021,7.008,148.435
C05273=1197.789,262.035,-64.603,-177.019,7.011,148.434
C05274=1197.784,262.284,-64.631,-177.016,7.012,148.434
C05275=1197.779,262.557,-64.661,-177.013,7.015,148.434
C05276=1197.775,262.829,-64.691,-177.010,7.018,148.434
C05277=1197.770,263.102,-64.721,-177.007,7.021,148.434
C05278=1197.765,263.375,-64.752,-177.004,7.024,148.434
C05279=1197.760,263.623,-64.779,-177.002,7.026,148.433
C05280=1197.756,263.872,-64.807,-177.000,7.028,148.433
C05281=1197.752,264.121,-64.834,-176.997,7.031,148.433
C05282=1197.747,264.368,-64.862,-176.995,7.033,148.433
C05283=1197.743,264.618,-64.889,-176.992,7.036,148.433
C05284=1197.739,264.865,-64.917,-176.989,7.038,148.433
C05285=1197.734,265.114,-64.944,-176.986,7.041,148.433
C05286=1197.731,265.363,-64.972,-176.984,7.043,148.433
C05287=1197.725,265.611,-65.000,-176.981,7.046,148.432
C05288=1197.721,265.859,-65.027,-176.979,7.048,148.432
C05289=1197.717,266.108,-65.056,-176.976,7.051,148.432
C05290=1197.712,266.356,-65.083,-176.974,7.053,148.432
C05291=1197.708,266.604,-65.110,-176.971,7.056,148.432
C05292=1197.704,266.853,-65.138,-176.969,7.058,148.432
C05293=1197.699,267.102,-65.166,-176.966,7.060,148.431
C05294=1197.695,267.349,-65.194,-176.963,7.063,148.431
C05295=1197.690,267.599,-65.221,-176.961,7.065,148.431
C05296=1197.686,267.847,-65.249,-176.958,7.068,148.431
C05297=1197.682,268.094,-65.277,-176.956,7.070,148.431
C05298=1197.677,268.344,-65.305,-176.953,7.073,148.431
C05299=1197.673,268.592,-65.333,-176.951,7.075,148.431
C05300=1197.669,268.840,-65.361,-176.948,7.078,148.431
C05301=1197.664,269.089,-65.388,-176.946,7.080,148.431
C05302=1197.659,269.337,-65.416,-176.943,7.083,148.430
C05303=1197.655,269.586,-65.445,-176.940,7.085,148.430
C05304=1197.651,269.833,-65.472,-176.938,7.088,148.430
C05305=1197.647,270.083,-65.500,-176.936,7.090,148.430
C05306=1197.642,270.331,-65.528,-176.932,7.093,148.430
C05307=1197.638,270.579,-65.556,-176.930,7.095,148.430
C05308=1197.634,270.827,-65.584,-176.928,7.098,148.430
C05309=1197.629,271.076,-65.612,-176.925,7.100,148.430
C05310=1197.625,271.325,-65.640,-176.922,7.103,148.429
C05311=1197.620,271.573,-65.668,-176.920,7.105,148.429
C05312=1197.616,271.821,-65.696,-176.917,7.108,148.429
C05313=1197.611,272.069,-65.724,-176.915,7.110,148.429
C05314=1197.608,272.318,-65.752,-176.912,7.113,148.429
C05315=1197.603,272.566,-65.781,-176.910,7.115,148.429
C05316=1197.598,272.814,-65.808,-176.907,7.118,148.429
C05317=1197.595,273.063,-65.837,-176.905,7.120,148.428
C05318=1197.589,273.311,-65.865,-176.902,7.123,148.428
C05319=1197.585,273.560,-65.892,-176.900,7.125,148.428
C05320=1197.580,273.808,-65.921,-176.897,7.128,148.428
C05321=1197.577,274.057,-65.949,-176.894,7.130,148.428
C05322=1197.572,274.305,-65.977,-176.892,7.133,148.428
C05323=1197.568,274.553,-66.005,-176.890,7.135,148.428
C05324=1197.563,274.801,-66.033,-176.887,7.138,148.428
C05325=1197.559,275.050,-66.062,-176.884,7.140,148.428
C05326=1197.554,275.298,-66.090,-176.882,7.143,148.428
C05327=1197.550,275.547,-66.118,-176.879,7.146,148.427
C05328=1197.546,275.796,-66.147,-176.877,7.148,148.427
C05329=1197.542,276.043,-66.175,-176.874,7.151,148.427
C05330=1197.538,276.292,-66.204,-176.871,7.153,148.427
C05331=1197.533,276.540,-66.232,-176.869,7.156,148.427
C05332=1197.529,276.788,-66.260,-176.867,7.158,148.427
C05333=1197.525,277.036,-66.288,-176.864,7.161,148.427
C05334=1197.520,277.285,-66.317,-176.861,7.163,148.427
C05335=1197.516,277.533,-66.345,-176.858,7.166,148.427
C05336=1197.511,277.782,-66.373,-176.856,7.168,148.427
C05337=1197.507,278.030,-66.401,-176.854,7.171,148.426
C05338=1197.503,278.278,-66.431,-176.851,7.173,148.426
C05339=1197.498,278.527,-66.459,-176.848,7.176,148.426
C05340=1197.494,278.775,-66.487,-176.846,7.179,148.426
C05341=1197.489,279.024,-66.516,-176.843,7.181,148.426
C05342=1197.485,279.272,-66.544,-176.841,7.184,148.426
C05343=1197.481,279.520,-66.573,-176.838,7.186,148.426
C05344=1197.477,279.769,-66.601,-176.835,7.189,148.426
C05345=1197.472,280.017,-66.630,-176.833,7.191,148.426
C05346=1197.467,280.266,-66.658,-176.831,7.194,148.426
C05347=1197.464,280.514,-66.687,-176.828,7.196,148.426
C05348=1197.459,280.762,-66.716,-176.826,7.199,148.425
C05349=1197.455,281.010,-66.744,-176.823,7.202,148.425
C05350=1197.450,281.258,-66.773,-176.820,7.204,148.425
C05351=1197.446,281.507,-66.802,-176.818,7.207,148.425
C05352=1197.442,281.755,-66.830,-176.816,7.209,148.425
C05353=1197.437,282.003,-66.859,-176.813,7.212,148.425
C05354=1197.433,282.252,-66.887,-176.810,7.214,148.425
C05355=1197.429,282.500,-66.916,-176.808,7.217,148.425
C05356=1197.424,282.748,-66.945,-176.805,7.220,148.425
C05357=1197.420,282.997,-66.973,-176.803,7.223,148.425
C05358=1197.416,283.245,-67.002,-176.800,7.226,148.425
C05359=1197.411,283.493,-67.031,-176.798,7.228,148.424
C05360=1197.407,283.742,-67.059,-176.795,7.231,148.424
C05361=1197.403,283.990,-67.089,-176.793,7.233,148.424
C05362=1197.398,284.238,-67.117,-176.790,7.236,148.424
C05363=1197.394,284.486,-67.146,-176.787,7.239,148.424
C05364=1197.390,284.735,-67.175,-176.785,7.241,148.424
C05365=1197.385,284.983,-67.204,-176.782,7.244,148.424
C05366=1197.381,285.231,-67.232,-176.780,7.246,148.424
C05367=1197.377,285.480,-67.262,-176.777,7.249,148.424
C05368=1197.372,285.728,-67.290,-176.774,7.252,148.424
C05369=1197.368,285.976,-67.319,-176.772,7.254,148.424
C05370=1197.364,286.224,-67.348,-176.769,7.257,148.424
C05371=1197.360,286.473,-67.377,-176.767,7.259,148.423
C05372=1197.356,286.721,-67.406,-176.765,7.262,148.423
C05373=1197.350,286.969,-67.435,-176.762,7.265,148.423
C05374=1197.346,287.218,-67.464,-176.760,7.267,148.423
C05375=1197.342,287.466,-67.494,-176.757,7.270,148.423
C05376=1197.338,287.714,-67.522,-176.754,7.272,148.423
C05377=1197.334,287.962,-67.551,-176.752,7.275,148.423
C05378=1197.329,288.210,-67.580,-176.749,7.278,148.423
C05379=1197.325,288.485,-67.612,-176.746,7.281,148.423
C05380=1197.320,288.760,-67.645,-176.744,7.284,148.423
C05381=1197.315,289.034,-67.677,-176.741,7.287,148.423
C05382=1197.310,289.308,-67.709,-176.738,7.290,148.423
C05383=1197.306,289.556,-67.738,-176.736,7.292,148.423
C05384=1197.302,289.805,-67.767,-176.733,7.295,148.423
C05385=1197.297,290.053,-67.796,-176.731,7.297,148.423
C05386=1197.293,290.301,-67.825,-176.728,7.300,148.422
C05387=1197.289,290.549,-67.855,-176.725,7.303,148.422
C05388=1197.284,290.798,-67.884,-176.723,7.305,148.422
C05389=1197.280,291.047,-67.913,-176.720,7.308,148.422
C05390=1197.276,291.295,-67.942,-176.718,7.311,148.422
C05391=1197.271,291.542,-67.972,-176.716,7.314,148.422
C05392=1197.267,291.791,-68.001,-176.713,7.317,148.422
C05393=1197.263,292.039,-68.030,-176.711,7.319,148.422
C05394=1197.258,292.287,-68.060,-176.708,7.322,148.422
C05395=1197.254,292.536,-68.089,-176.705,7.325,148.422
C05396=1197.250,292.784,-68.118,-176.703,7.327,148.422
C05397=1197.246,293.033,-68.148,-176.700,7.330,148.422
C05398=1197.241,293.280,-68.177,-176.697,7.333,148.422
C05399=1197.237,293.528,-68.206,-176.695,7.335,148.422
C05400=1197.232,293.777,-68.236,-176.693,7.338,148.422
C05401=1197.228,294.025,-68.265,-176.690,7.341,148.422
C05402=1197.224,294.273,-68.294,-176.688,7.343,148.422
C05403=1197.220,294.521,-68.324,-176.685,7.346,148.422
C05404=1197.216,294.770,-68.353,-176.683,7.348,148.422
C05405=1197.211,295.018,-68.383,-176.680,7.351,148.422
C05406=1197.207,295.266,-68.412,-176.677,7.354,148.422
C05407=1197.203,295.515,-68.442,-176.675,7.357,148.421
C05408=1197.198,295.762,-68.471,-176.673,7.360,148.421
C05409=1197.194,296.010,-68.500,-176.670,7.363,148.421
C05410=1197.189,296.259,-68.530,-176.668,7.365,148.421
C05411=1197.185,296.507,-68.560,-176.665,7.368,148.421
C05412=1197.181,296.755,-68.589,-176.662,7.371,148.421
C05413=1197.177,297.004,-68.619,-176.660,7.373,148.421
C05414=1197.173,297.251,-68.649,-176.657,7.376,148.421
C05415=1197.169,297.500,-68.678,-176.655,7.379,148.421
C05416=1197.164,297.748,-68.708,-176.653,7.381,148.421
C05417=1197.160,297.997,-68.738,-176.650,7.384,148.421
C05418=1197.155,298.245,-68.767,-176.647,7.387,148.421
C05419=1197.151,298.493,-68.797,-176.645,7.389,148.421
C05420=1197.147,298.741,-68.827,-176.642,7.392,148.421
C05421=1197.143,298.989,-68.856,-176.640,7.395,148.421
C05422=1197.138,299.238,-68.886,-176.638,7.398,148.421
C05423=1197.134,299.486,-68.916,-176.635,7.401,148.421
C05424=1197.130,299.734,-68.945,-176.632,7.404,148.421
C05425=1197.126,299.982,-68.975,-176.630,7.406,148.421
C05426=1197.121,300.230,-69.005,-176.627,7.409,148.421
C05427=1197.117,300.479,-69.035,-176.625,7.412,148.421
C05428=1197.113,300.726,-69.065,-176.623,7.414,148.421
C05429=1197.109,300.974,-69.095,-176.620,7.417,148.421
C05430=1197.104,301.223,-69.125,-176.618,7.420,148.421
C05431=1197.100,301.471,-69.154,-176.615,7.423,148.421
C05432=1197.096,301.719,-69.184,-176.613,7.426,148.421
C05433=1197.091,301.968,-69.214,-176.610,7.429,148.421
C05434=1197.087,302.215,-69.244,-176.608,7.431,148.421
C05435=1197.083,302.463,-69.274,-176.605,7.434,148.421
C05436=1197.078,302.712,-69.304,-176.602,7.437,148.421
C05437=1197.074,302.960,-69.334,-176.600,7.439,148.421
C05438=1197.070,303.208,-69.364,-176.598,7.442,148.421
C05439=1197.065,303.456,-69.394,-176.595,7.445,148.421
C05440=1197.061,303.704,-69.424,-176.593,7.447,148.421
C05441=1197.057,303.952,-69.453,-176.591,7.451,148.421
C05442=1197.053,304.201,-69.484,-176.588,7.454,148.421
C05443=1197.049,304.449,-69.514,-176.585,7.457,148.421
C05444=1197.044,304.697,-69.545,-176.583,7.459,148.421
C05445=1197.040,304.946,-69.574,-176.580,7.462,148.421
C05446=1197.036,305.193,-69.604,-176.578,7.465,148.421
C05447=1197.031,305.442,-69.634,-176.576,7.467,148.421
C05448=1197.027,305.689,-69.664,-176.573,7.470,148.421
C05449=1197.023,305.937,-69.695,-176.570,7.473,148.421
C05450=1197.018,306.186,-69.725,-176.568,7.476,148.421
C05451=1197.014,306.434,-69.755,-176.566,7.479,148.421
C05452=1197.010,306.683,-69.785,-176.563,7.482,148.421
C05453=1197.006,306.931,-69.816,-176.560,7.485,148.421
C05454=1197.002,307.178,-69.846,-176.558,7.487,148.421
C05455=1196.997,307.427,-69.876,-176.556,7.490,148.421
C05456=1196.993,307.674,-69.906,-176.553,7.493,148.421
C05457=1196.988,307.923,-69.936,-176.551,7.495,148.421
C05458=1196.984,308.171,-69.967,-176.548,7.498,148.421
C05459=1196.980,308.419,-69.998,-176.546,7.501,148.421
C05460=1196.976,308.667,-70.028,-176.544,7.504,148.421
C05461=1196.971,308.916,-70.058,-176.541,7.507,148.421
C05462=1196.967,309.163,-70.088,-176.538,7.510,148.421
C05463=1196.963,309.411,-70.119,-176.536,7.513,148.421
C05464=1196.959,309.659,-70.148,-176.534,7.515,148.421
C05465=1196.955,309.908,-70.179,-176.531,7.518,148.421
C05466=1196.950,310.156,-70.210,-176.528,7.521,148.421
C05467=1196.946,310.404,-70.240,-176.526,7.523,148.421
C05468=1196.942,310.652,-70.271,-176.524,7.526,148.421
C05469=1196.937,310.900,-70.301,-176.521,7.530,148.421
C05470=1196.933,311.149,-70.332,-176.519,7.533,148.421
C05471=1196.929,311.397,-70.362,-176.517,7.535,148.421
C05472=1196.925,311.644,-70.393,-176.514,7.538,148.421
C05473=1196.920,311.892,-70.423,-176.512,7.541,148.421
C05474=1196.917,312.140,-70.454,-176.509,7.543,148.421
C05475=1196.912,312.389,-70.484,-176.507,7.546,148.421
C05476=1196.907,312.637,-70.515,-176.504,7.549,148.421
C05477=1196.904,312.885,-70.545,-176.501,7.552,148.421
C05478=1196.900,313.133,-70.576,-176.500,7.555,148.421
